(**********************Pointing************************)	
	(*ActAmbTemp_East:LREAL;
	ActAmbTemp_South:LREAL;
	AmbTempCorrVal_1:LREAL;
	AmbTempCorrVal_2:LREAL;
	TiltXRaw_One:LREAL;
	TiltYRaw_One:LREAL;
	TiltXArcsec_One:LREAL;
	TiltYArcsec_One: BOOL;
	TiltXFilt_One:LREAL;
	TiltYFilt_One:LREAL;
	TiltTemp_One:LREAL;
	TiltXRaw_Two:LREAL;
	TiltYRaw_Two:LREAL;
	TiltXArcsec_Two:LREAL;
	TiltYArcsec_Two: BOOL;
	TiltXFilt_Two:LREAL;
	TiltYFilt_Two:LREAL;
	TiltTemp_Two:LREAL;
	TiltCorrVal_Az:LREAL;
	TiltCorrVal_EL:LREAL;
	PmCorrVal_Az: BOOL;
	PmCorrVal_EL: BOOL;
	StaticCorrActive:BOOL;
	TiltCorrActive:BOOL;
	Pointing_TiltOn:UINT;
	TempCorrActive:BOOL;
	BandForCorr:UINT;*)
	Pointing_TiltOn:UINT;
(**************************Tracking********************************)
(*	tr_initOk:BOOL;(*Tracking function program is initialized and ready for operation*)
	tr_valid:BOOL;(*The tracking controller’s output is within the position ranges of the dish structure.*)
	tr_Table_error:BOOL;(*The table reports an error *)
	tr_obj_valid:BOOL;(*Tracking object has valid tracking data.*)
	tr_selFIy:BOOL;(*FIynomial tracking selected as source*)
	act_statOffset_value_Xel:LREAL;(*Actual azimuth static offset*)
	act_statOffset_value_El:LREAL;(*Elevation azimuth static offset*)
	p_desired_AZ:LREAL;(*Azimuth position output of the Tracking Controller*)
	p_desired_EL:LREAL;(*Elevation position output of the Tracking Controller*)
	tr_TimeRemaining:LREAL;(*Time till the last point in the track table is reached*)
	OnSourceDev:LREAL;(*Actual calculated “On Sky” rms tracking error.*) *)
(*********Read parameteers*******)
	AxRef:ARRAY[1..5] OF AXIS_REF;
	P_shape_value:ARRAY[1..5] OF LREAL;
	V_shape_value:ARRAY[1..5] OF LREAL;
	V_act_value:ARRAY[1..5] OF LREAL;
	r_write_position_az: LREAL; // Used internally for interpolator and pointing model calculations
    r_write_position_az_out: LREAL; (*the position written to the virvual azimuth axis*)
	r_write_position_el: LREAL; // Used internally for interpolator and pointing model calculations
    r_write_position_el_out: LREAL;(*the position written to the virvual elevation axis*)
	r_write_position_FI: LREAL;(*the position written to the virvual FeedIndexer axis*)
	r_write_position_FI_out: LREAL;(*the position written to the virvual FeedIndexer axis*)
	
END_VAR

VAR_GLOBAL RETAIN PERSISTENT
	R_total_distance_AZ:LREAL;
	R_total_distance_EL_deg:LREAL;
	R_total_distance_EL_m:LREAL;
	R_total_distance_FI:LREAL;
	
	LeapSecPTP: UINT :=37;    // Storage for Leap seconds 
	
END_VAR

// IndraMotionMlc1/Application/POUs/Motion/P_Position_and_MJD
(*The program is built for calculating the position of real axis, virtual axis and the MJD time,
and writing software limit of azimuth *)
PROGRAM P_Position_and_MJD
VAR
(*With the function block "MB_WriteRealParameter" you can write a defined value to the parameter belonging to the parameter number*)
	fb_write_negative_a: MB_WriteRealParameter;
	fb_write_negative_s: MB_WriteRealParameter;
	fb_write_positive_a: MB_WriteRealParameter;
	fb_write_positive_s: MB_WriteRealParameter;
(*the blink function block is for triggering MB_WriteRealParameter function block*)
	fb_blink_1: BLINK;
	fb_blink_2: BLINK;
	fb_blink_3: BLINK;
	fb_blink_4: BLINK;
(*the value is written to MB_WriteRealParameter*)
	r_negative_limit: REAL;
	r_positive_limit: REAL;
(*the elevation limit control*)
	fb_blink_diagnos_el: BLINK;
	fb_diagnose_el: MB_ReadStringParameter;
	str_diagnose_el: STRING;
	fb_blink_5: BLINK;
	fb_blink_6: BLINK;
	fb_write_negative_el: MB_WriteRealParameter;
	fb_write_positive_el: MB_WriteRealParameter;
	r_limit_el_up: REAL;
	r_limit_el_down: REAL;
	b_limit_up_el: BOOL;
	b_limit_down_el: BOOL;
	rtrig_set_limit_up: R_TRIG;
	rtrig_set_limit_down: R_TRIG;
	fb_blink_7: BLINK;
	fb_write_91_az1: MB_WriteRealParameter;
	fb_blink_8: BLINK;
	fb_blink_9: BLINK;
	fb_blink_10: BLINK;
	fb_blink_11: BLINK;
	fb_write_91_az2: MB_WriteRealParameter;
	fb_write_91_el1: MB_WriteRealParameter;
	fb_write_91_el2: MB_WriteRealParameter;
	fb_write_91_FI: MB_WriteRealParameter;
	fb_blink_12: BLINK;
	fb_write_91_FI2: MB_WriteRealParameter;
	r_pos_FI_1: REAL;
	i_counter_hr: BOOL;
	rtrig_hr:R_TRIG;
	
	fb_blink_111: BLINK;
	fb_write_negative_a_v: MB_WriteRealParameter;
	fb_blink_1_v: BLINK;
	fb_blink_2_v: BLINK;
	fb_write_negative_s_v: MB_WriteRealParameter;
	fb_blink_3_v: BLINK;
	fb_write_positive_a_v: MB_WriteRealParameter;
	
	temp_a:LREAL:=3135.4451;
	temp_b:LREAL:=3013.785;	
	temp_c:LREAL;
	r_pos_az_org :LREAL;
	r_pos_az_v_org :LREAL;
	r_pos_el_org:LREAL;
	r_pos_el_v_org:LREAL;

	fb_real_drive3_s51: MB_ReadRealParameter;
	r_pos_motor3_1: REAL;
	
	i_overlop:BOOL;
	rtrig_overlop:R_TRIG;
	
	
	DeltaB_temp: LREAL;
	
	B_TEMP: LREAL;
	
	MB_AxisDistanceAccumulator_2: MB_AxisDistanceAccumulator;
	bDisenable1: BOOL;
	test_1: LREAL;
	test_2: LREAL;
	test_old: LREAL;
	normal_count:DINT:=995;
	low_count:DINT:=9995;
	fast_count:DINT:=9995;
	i_change_sign_count:DINT;
	r_threshold:REAL;
END_VAR
VAR RETAIN
	r_last_position_az: REAL:=1;
	l_control:LREAL;
	a_control:REAL:=3035.4;
	b_control:REAL:=3035.1;
	b_motor_count:DINT:=0;
	b_sign_delay:BOOL:=0;
	b_sign_delay_count:DINT:=0;
	r_test_value:LREAL;
	i_test_value:DINT:=0;
	fb_read_source_code_3: MB_ReadParameter;
	r_source_code_3: DINT;
	r_source_to_elevation: LREAL;
END_VAR

 	//axisdata[7].rActualPosition_i;
r_source_to_elevation:=(DINT_TO_LREAL(r_source_code_3)/536870912)*360.0-64.812477;

	MB_AxisDistanceAccumulator_2(
	Enable:= bDisenable1, 
	TotalDistance:= 1000000, 
	InOperation=> , 
	Error=> , 
	ErrorID=> , 
	ErrorIdent=> , 
	DistanceReached=> , 
	AccumulatedDistance=> r_length_Distance_1, 
	Axis:= Drive3);
	
	IF	r_pos_motor3<0.01 AND r_pos_motor3>=0 THEN
	i_overlop:=TRUE;
	ELSE
	i_overlop:=FALSE;
	END_IF	
	rtrig_overlop(clk:=i_overlop);
	IF rtrig_overlop.Q=TRUE THEN
	b_motor_count:=b_motor_count+1;
	END_IF
		
	l_control:=SQRT(a_control*a_control+b_control*b_control-2*a_control*b_control*COS(deg2rad(112.0255-ML_Base.AxisData[3].rActualPosition_i)))-1151;
//	
//	temp_c:= SQRT(temp_a*temp_a + temp_b*temp_b-2*temp_a*temp_b*COS((115.5-r_pos_el_v)*3.1415926/180.0));
//	gear_ratio:=temp_a*temp_b*SIN((115.5-r_pos_el_v)*3.1415926/180.0)/temp_c*6.0*168.0/25.0/180.0*3.1415926;
	
	

(*<<time1<<<<<<<<<<<<<<<<<<<<<<<<<<<<<< real position of azimuth elevation and FeedIndexer>>>>>>>>>>>>>>>>>>>>>>>>>>>>>>>>*)
(*the azimuth position is judged by zone signal*)

	IF axisdata[1].Axis_Inbb=TRUE THEN	
		//r_pos_az_org:=axisdata[1].rActualPosition_i;
		//r_pos_az_1:=r_pos_az_org+C1+C3*SIN((r_pos_az_org-C4)*3.1415926/180)*TAN(r_pos_el_org*3.1415926/180)+C5*TAN(r_pos_el_org*3.1415926/180)+C6/COS(r_pos_el_org*3.1415926/180);		
	//	r_pos_az_modify:=r_pos_az_1;
	    r_pos_az_modify:=axisdata[1].rActualPosition_i;
		IF r_pos_az_1>=360.0 THEN 
			r_pos_az_modify:=r_pos_az_1-360.00;
		END_IF
		IF r_pos_az_1<0.0 THEN 
			r_pos_az_modify:=r_pos_az_1+360.00;
		END_IF
			
	END_IF;		
		(*IF b_zone_az=FALSE AND axisdata[1].rActualPosition_i>75 AND axisdata[1].rActualPosition_i<360 THEN
			r_pos_az:=axisdata[1].rActualPosition_i-360;
			r_pos_az_v:=axisdata[1].rActualPosition_i-360;
//		ELSIF axisdata[1].rActualPosition_i>299 THEN
	//		r_pos_az:=axisdata[1].rActualPosition_i-360;
//			r_pos_az_v:=axisdata[1].rActualPosition_i-360;
        ELSE
        r_pos_az:=axisdata[1].rActualPosition_i;
		r_pos_az_v:=axisdata[1].rActualPosition_i;
		END_IF;*)
        r_pos_az:=axisdata[1].rActualPosition_i;
		r_pos_az_v:=axisdata[7].rActualPosition_i;
	//	END_IF;
   IF gc_b_sim_on THEN
	IF ABS (r_pos_az_v ) = 360 THEN	
	r_pos_az:=0.0000;
	r_pos_az_v := 0.0000;
	END_IF
   END_IF
	
	//angleerror := axisdata[1].rActualPosition_i - axisdata[2].rActualPosition_i;

	AZ_encoder_last:=r_pos_az_v;
	
	IF axisdata[5].rActualPosition_i < 180 THEN
		r_pos_Fi:=axisdata[5].rActualPosition_i;
	    r_pos_Fi_v:=axisdata[5].rActualPosition_i;
	ELSE
		r_pos_Fi:=axisdata[5].rActualPosition_i-360;
	    r_pos_Fi_v:=axisdata[5].rActualPosition_i-360;
	END_IF
	FI_encoder_last:=r_pos_fi_v;
	
//r_pos_el_org:=axisdata[3].rActualPosition_i;
//r_pos_el_1:=r_pos_el_org+C2+C3*COS((r_pos_az_org-C4)*3.1415926/180)+C7*COS(r_pos_el_org*3.1415926/180)+0;	
//r_pos_el_modify	:=r_pos_el_1;
r_pos_el:=axisdata[3].rActualPosition_i;
//r_pos_el:=r_source_to_elevation;
r_pos_el_v:=axisdata[3].rActualPosition_i;
(* From SKA063 project
r_pos_el:=ML_Base.AxisData[11].rActualPosition_i;
r_pos_el_v:=ML_Base.AxisData[11].rActualPosition_i; *)

(*<<<<<<<<<<<<<<<<<<<<<<<<<<<<<<<<<<<<<<<<<<<<<<<<<<<calculation for MJD >>>>>>>>>>>>>>>>>>>>>>>>>>>>>>>>>>>>>>>*)
(*the definition of MJD is shown in the global variables*)
(*the module of v_time_master axis is 360,so that it take 6minuts to run one cycle*)
IF	axisdata[10].rActualPosition_i<0.01 AND axisdata[10].rActualPosition_i>=0 THEN
	i_counter_hr:=TRUE;
ELSE
	i_counter_hr:=FALSE;
END_IF	
rtrig_hr(clk:=i_counter_hr);
IF rtrig_hr.Q=TRUE THEN
	i_num_quarter:=i_num_quarter+1;
END_IF
IF i_num_quarter=240 THEN
	i_num_quarter:=0;
	di_MJD_day:=di_MJD_day+1;
END_IF

//lr_MJD_current:=TO_REAL(di_MJD_day)+(360*TO_REAL(i_num_quarter)+axisdata[10].rActualPosition_i)/86400+1.0/3.0; // Sets MJD to Beijing time
lr_MJD_current:=TO_REAL(di_MJD_day)+(360*TO_REAL(i_num_quarter)+axisdata[10].rActualPosition_i)/86400;
lr_TAIoffset_current:= (lr_MJD_Current-gc_SKAEpochMJD)*86400+(time_cds.Status.LeapSecPTP); // Minus 10s if you want to correlate to a unix timestamp


(*<<<<<<<<<<<<<<<<<calculate the following error of trajectory>>>>>>>>>>>>>>>>>>>*)

IF ABS(r_vel_EL)>=0.5 THEN
	r_threshold:=0.25;
ELSE 
	r_threshold:=0.15;
END_IF

IF b_open_channel_az AND b_open_channel_el THEN
//IF ABS(lr_MJD_current-track_table[i_start].MJD-0.0000000254)*86400<=0.0005 AND b_sign_delay=0 THEN
	IF ABS(lr_TAIoffset_current-track_table[i_start].TAIoffset-0.0022)<=0.0005 AND b_sign_delay=0 THEN
	b_sign_delay:=1;
//	r_test_value:=0;
	i_test_value:=0;
	r_track_error[1]:=track_table[i_start].Azimuth-r_pos_az;
	
(*   For Elevation orientation axis

	r_track_error[2]:=track_table[i_start].Elevation_ori+r_offset_el_program-r_pos_el;
   IF ABS(r_track_error[2])<r_threshold THEN
		test_1:=Encoder_to_motor(track_table[i_start].Elevation_ori)-Encoder_to_motor(track_table[i_start].Elevation_ori-r_track_error[2]);
		test_2:=Encoder_to_motor(track_table[i_start].Elevation_ori)-Encoder_to_motor(track_table[i_start].Elevation_ori+r_track_error[2]);
//		test_3:=test_1+test_old;
	ELSE
		test_1:=0;
		test_2:=0;
		r_compensation_abs:=0;
		test_old:=0;
	END_IF *)
	
END_IF
	IF b_sign_delay =1 THEN

	i_test_value:=i_test_value+1;
	
	IF i_test_value>995 THEN 
		r_test_value:=r_compensation_abs;
	ELSE
		r_test_value:=r_compensation_abs+test_1/995;
	END_IF
		r_compensation_abs:=r_test_value;
		
	END_IF
		
	END_IF

IF b_sign_delay =1 THEN 
	b_sign_delay_count:=b_sign_delay_count+1;
END_IF

IF ABS(r_vel_EL)<0.002 THEN
	i_change_sign_count:=9995;
ELSIF ABS(r_vel_EL)>0.6 AND ABS(r_vel_EL)<0.8 THEN
	i_change_sign_count:=9995;
ELSIF ABS(r_vel_EL)>=0.8 THEN
	i_change_sign_count:=12995;	
ELSE 
	i_change_sign_count:=normal_count;	
END_IF




IF b_sign_delay_count>i_change_sign_count THEN
	b_sign_delay_count:=0;
	b_sign_delay:=0;
END_IF




IF b_off_write=TRUE THEN
	r_limit_s91:=11;
ELSE
	r_limit_s91:=1.4;
END_IF;
(*<<<<<<<<<<<<<<<<<<the azimuth limit control>>>>>>>>>>>>>>>>>>>>*)
IF (r_pos_az<-250) OR (r_pos_az>250) THEN
(*the range of azimuth is -179~359*)
	//r_negative_limit:=89;
	//r_positive_limit:=271;
	r_negative_limit:=-275;
	r_positive_limit:=275;
ELSE
	//r_negative_limit:=0;
	//r_positive_limit:=360;
	r_negative_limit:=-275;
	r_positive_limit:=275;
END_IF;
(*
(*<<<<<<<<<<<<<<<<<<<<<<<<<the elevation limit control>>>>>>>>>>>>>>>>>>>>>>>*)
IF str_diagnose_el='F6029 ' THEN
	b_limit_up_el:=TRUE;
ELSE
	b_limit_up_el:=FALSE;
END_IF
rtrig_set_limit_up(clk:=b_limit_up_el);
IF rtrig_set_limit_up.Q=TRUE THEN
	r_limit_el_up:=90.05;
END_IF
IF r_pos_el <=90.1 THEN
	r_limit_el_up:=90.15;
END_IF

IF str_diagnose_el='F6030 ' THEN
	b_limit_down_el:=TRUE;
ELSE
	b_limit_down_el:=FALSE;
END_IF
rtrig_set_limit_down(clk:=b_limit_down_el);
IF rtrig_set_limit_down.Q=TRUE THEN
	r_limit_el_down:=14.7;
END_IF
IF r_pos_el >=14.65 THEN
	r_limit_el_down:=14.6;
END_IF
*)



//P_Position_and_MJD.A_Write_Limit_Value();lr_TAIoffset_current
//Time Sensitive pointing data
Time_cds.Status.TAIOffset:=lr_TAIoffset_current;
IF gc_b_sim_on THEN 
	IF r_pos_az = -360 THEN
		r_pos_az:= 0;
	END_IF

END_IF

Azimuth.Status.p_Act:=pointing.Status.TotalPointCorr_Az/gc_lr_arcsec2deg+r_pos_az;
Azimuth.Status.p_Enc:=r_pos_az;
Elevation.Status.p_Act:=pointing.Status.TotalPointCorr_El/gc_lr_arcsec2deg+r_pos_el;
Elevation.Status.p_Enc:=r_pos_el;

Pointing.Status.CurrentPointing[0]:= Time_cds.Status.TAIoffset;
Pointing.Status.CurrentPointing[1]:= Azimuth.Status.p_Act;
Pointing.Status.CurrentPointing[2]:= Elevation.Status.p_Act;
Pointing.Status.CurrentPointing[3]:= Azimuth.Status.p_Enc;
Pointing.Status.CurrentPointing[4]:= Elevation.Status.p_Enc;
Pointing.Status.CurrentPointing[5]:= pointing.Status.TiltCorrVal_Az;
Pointing.Status.CurrentPointing[6]:= pointing.Status.TiltCorrVal_El;

ACTION A_Write_Limit_Value:
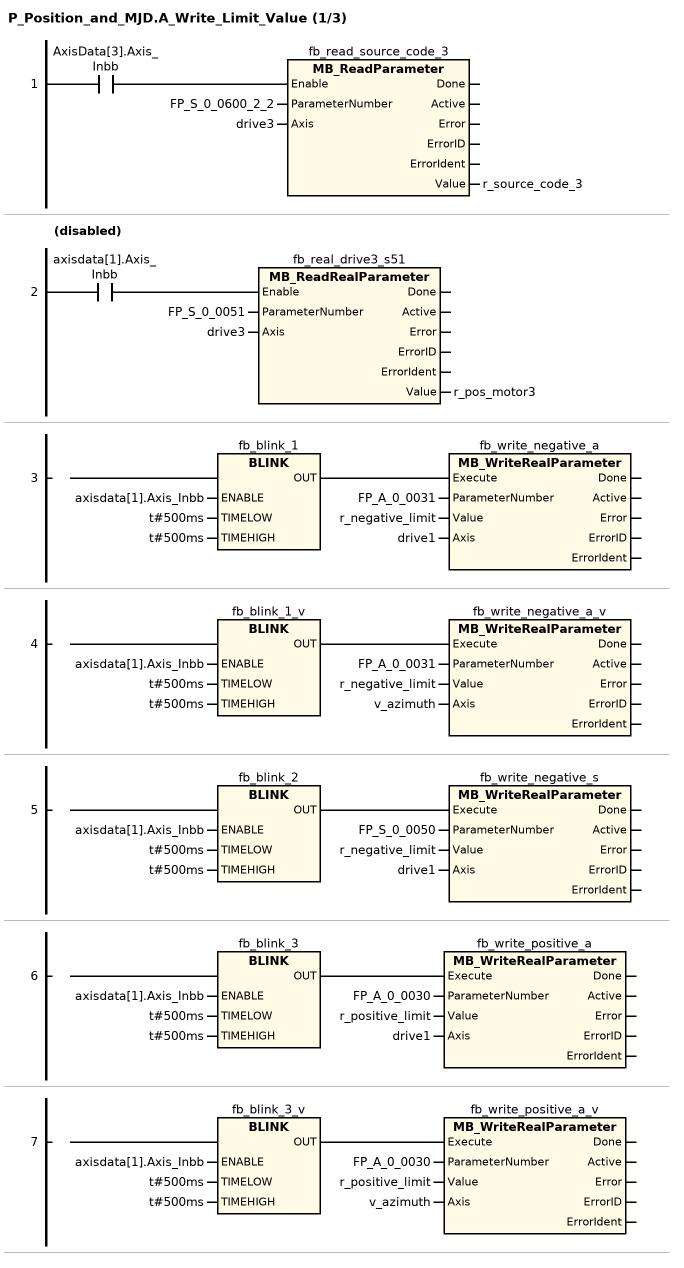
// NETWORK 1
fb_read_source_code_3(
    Enable := AxisData[3].Axis_Inbb,
    ParameterNumber := FP_S_0_0600_2_2,
    Axis := drive3,
    Value => r_source_code_3); // MB_ReadParameter

// NETWORK 2 (disabled)
//   FP_S_0_0051: Position limit value, negative
//   drive3: the value is written to MB_WriteRealParameter
// fb_real_drive3_s51(
//     Enable := axisdata[1].Axis_Inbb,
//     ParameterNumber := FP_S_0_0051,
//     Axis := drive3,
//     Value => r_pos_motor3); // MB_ReadRealParameter

// NETWORK 3
//   fb_write_negative_a: With the function block "MB_WriteRealParameter" you can write a defined value to the parameter belonging to the parameter number
//   fb_blink_1: the blink function block is for triggering MB_WriteRealParameter function block
//   axisdata[1].Axis_Inbb: A-0-0021.13 -RD- Axis is ready for power to the amplifier (bb)
//   FP_A_0_0031: Position limit value, negative
//   r_negative_limit: the value is written to MB_WriteRealParameter
//   drive1: Real axis "Drive1" with axis number 1
fb_blink_1(ENABLE := axisdata[1].Axis_Inbb, TIMELOW := t#500ms, TIMEHIGH := t#500ms); // BLINK
fb_write_negative_a(
    Execute := fb_blink_1.OUT,
    ParameterNumber := FP_A_0_0031,
    Value := r_negative_limit,
    Axis := drive1); // MB_WriteRealParameter

// NETWORK 4
//   axisdata[1].Axis_Inbb: A-0-0021.13 -RD- Axis is ready for power to the amplifier (bb)
//   FP_A_0_0031: Position limit value, negative
//   r_negative_limit: the value is written to MB_WriteRealParameter
//   v_azimuth: Virtual axis "v_azimuth" with axis number 7
fb_blink_1_v(ENABLE := axisdata[1].Axis_Inbb, TIMELOW := t#500ms, TIMEHIGH := t#500ms); // BLINK
fb_write_negative_a_v(
    Execute := fb_blink_1_v.OUT,
    ParameterNumber := FP_A_0_0031,
    Value := r_negative_limit,
    Axis := v_azimuth); // MB_WriteRealParameter

// NETWORK 5
//   axisdata[1].Axis_Inbb: A-0-0021.13 -RD- Axis is ready for power to the amplifier (bb)
//   FP_S_0_0050: Negative position limit value
//   r_negative_limit: the value is written to MB_WriteRealParameter
//   drive1: Real axis "Drive1" with axis number 1
fb_blink_2(ENABLE := axisdata[1].Axis_Inbb, TIMELOW := t#500ms, TIMEHIGH := t#500ms); // BLINK
fb_write_negative_s(
    Execute := fb_blink_2.OUT,
    ParameterNumber := FP_S_0_0050,
    Value := r_negative_limit,
    Axis := drive1); // MB_WriteRealParameter

// NETWORK 6
//   axisdata[1].Axis_Inbb: A-0-0021.13 -RD- Axis is ready for power to the amplifier (bb)
//   FP_A_0_0030: Position limit value, positive
//   drive1: Real axis "Drive1" with axis number 1
fb_blink_3(ENABLE := axisdata[1].Axis_Inbb, TIMELOW := t#500ms, TIMEHIGH := t#500ms); // BLINK
fb_write_positive_a(
    Execute := fb_blink_3.OUT,
    ParameterNumber := FP_A_0_0030,
    Value := r_positive_limit,
    Axis := drive1); // MB_WriteRealParameter

// NETWORK 7
//   axisdata[1].Axis_Inbb: A-0-0021.13 -RD- Axis is ready for power to the amplifier (bb)
//   FP_A_0_0030: Position limit value, positive
//   v_azimuth: Virtual axis "v_azimuth" with axis number 7
fb_blink_3_v(ENABLE := axisdata[1].Axis_Inbb, TIMELOW := t#500ms, TIMEHIGH := t#500ms); // BLINK
fb_write_positive_a_v(
    Execute := fb_blink_3_v.OUT,
    ParameterNumber := FP_A_0_0030,
    Value := r_positive_limit,
    Axis := v_azimuth); // MB_WriteRealParameter

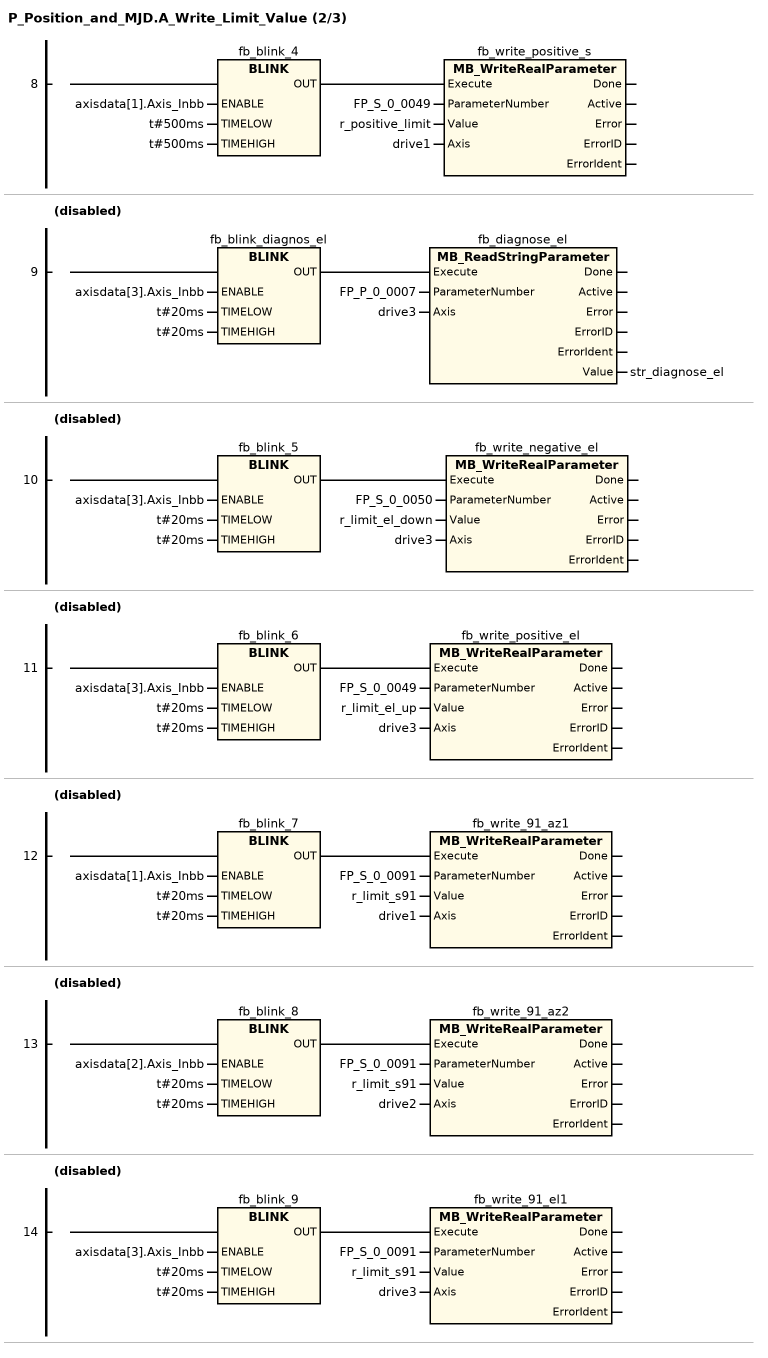
// NETWORK 8
//   axisdata[1].Axis_Inbb: A-0-0021.13 -RD- Axis is ready for power to the amplifier (bb)
//   FP_S_0_0049: Positive position limit value
//   drive1: Real axis "Drive1" with axis number 1
fb_blink_4(ENABLE := axisdata[1].Axis_Inbb, TIMELOW := t#500ms, TIMEHIGH := t#500ms); // BLINK
fb_write_positive_s(
    Execute := fb_blink_4.OUT,
    ParameterNumber := FP_S_0_0049,
    Value := r_positive_limit,
    Axis := drive1); // MB_WriteRealParameter

// NETWORK 9 (disabled)
//   fb_blink_diagnos_el: the elevation limit control
//   axisdata[3].Axis_Inbb: A-0-0021.13 -RD- Axis is ready for power to the amplifier (bb)
//   FP_P_0_0007: Display text of diagnostic message
//   drive3: Real axis "Drive3" with axis number 3
// fb_blink_diagnos_el(ENABLE := axisdata[3].Axis_Inbb, TIMELOW := t#20ms, TIMEHIGH := t#20ms); // BLINK
// fb_diagnose_el(
//     Execute := fb_blink_diagnos_el.OUT,
//     ParameterNumber := FP_P_0_0007,
//     Axis := drive3,
//     Value => str_diagnose_el); // MB_ReadStringParameter

// NETWORK 10 (disabled)
//   axisdata[3].Axis_Inbb: A-0-0021.13 -RD- Axis is ready for power to the amplifier (bb)
//   FP_S_0_0050: Negative position limit value
//   drive3: Real axis "Drive3" with axis number 3
// fb_blink_5(ENABLE := axisdata[3].Axis_Inbb, TIMELOW := t#20ms, TIMEHIGH := t#20ms); // BLINK
// fb_write_negative_el(
//     Execute := fb_blink_5.OUT,
//     ParameterNumber := FP_S_0_0050,
//     Value := r_limit_el_down,
//     Axis := drive3); // MB_WriteRealParameter

// NETWORK 11 (disabled)
//   axisdata[3].Axis_Inbb: A-0-0021.13 -RD- Axis is ready for power to the amplifier (bb)
//   FP_S_0_0049: Positive position limit value
//   drive3: Real axis "Drive3" with axis number 3
// fb_blink_6(ENABLE := axisdata[3].Axis_Inbb, TIMELOW := t#20ms, TIMEHIGH := t#20ms); // BLINK
// fb_write_positive_el(
//     Execute := fb_blink_6.OUT,
//     ParameterNumber := FP_S_0_0049,
//     Value := r_limit_el_up,
//     Axis := drive3); // MB_WriteRealParameter

// NETWORK 12 (disabled)
//   axisdata[1].Axis_Inbb: A-0-0021.13 -RD- Axis is ready for power to the amplifier (bb)
//   FP_S_0_0091: Bipolar velocity limit value
//   drive1: Real axis "Drive1" with axis number 1
// fb_blink_7(ENABLE := axisdata[1].Axis_Inbb, TIMELOW := t#20ms, TIMEHIGH := t#20ms); // BLINK
// fb_write_91_az1(
//     Execute := fb_blink_7.OUT,
//     ParameterNumber := FP_S_0_0091,
//     Value := r_limit_s91,
//     Axis := drive1); // MB_WriteRealParameter

// NETWORK 13 (disabled)
//   axisdata[2].Axis_Inbb: A-0-0021.13 -RD- Axis is ready for power to the amplifier (bb)
//   FP_S_0_0091: Bipolar velocity limit value
//   drive2: Real axis "Drive2" with axis number 2
// fb_blink_8(ENABLE := axisdata[2].Axis_Inbb, TIMELOW := t#20ms, TIMEHIGH := t#20ms); // BLINK
// fb_write_91_az2(
//     Execute := fb_blink_8.OUT,
//     ParameterNumber := FP_S_0_0091,
//     Value := r_limit_s91,
//     Axis := drive2); // MB_WriteRealParameter

// NETWORK 14 (disabled)
//   axisdata[3].Axis_Inbb: A-0-0021.13 -RD- Axis is ready for power to the amplifier (bb)
//   FP_S_0_0091: Bipolar velocity limit value
//   drive3: Real axis "Drive3" with axis number 3
// fb_blink_9(ENABLE := axisdata[3].Axis_Inbb, TIMELOW := t#20ms, TIMEHIGH := t#20ms); // BLINK
// fb_write_91_el1(
//     Execute := fb_blink_9.OUT,
//     ParameterNumber := FP_S_0_0091,
//     Value := r_limit_s91,
//     Axis := drive3); // MB_WriteRealParameter

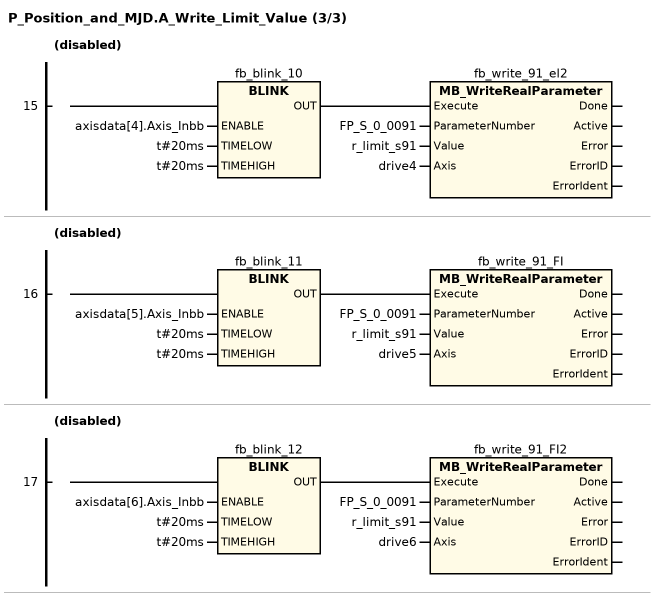
// NETWORK 15 (disabled)
//   axisdata[4].Axis_Inbb: A-0-0021.13 -RD- Axis is ready for power to the amplifier (bb)
//   FP_S_0_0091: Bipolar velocity limit value
//   drive4: Real axis "Drive4" with axis number 4
// fb_blink_10(ENABLE := axisdata[4].Axis_Inbb, TIMELOW := t#20ms, TIMEHIGH := t#20ms); // BLINK
// fb_write_91_el2(
//     Execute := fb_blink_10.OUT,
//     ParameterNumber := FP_S_0_0091,
//     Value := r_limit_s91,
//     Axis := drive4); // MB_WriteRealParameter

// NETWORK 16 (disabled)
//   axisdata[5].Axis_Inbb: A-0-0021.13 -RD- Axis is ready for power to the amplifier (bb)
//   FP_S_0_0091: Bipolar velocity limit value
//   drive5: Real axis "Drive5" with axis number 5
// fb_blink_11(ENABLE := axisdata[5].Axis_Inbb, TIMELOW := t#20ms, TIMEHIGH := t#20ms); // BLINK
// fb_write_91_FI(
//     Execute := fb_blink_11.OUT,
//     ParameterNumber := FP_S_0_0091,
//     Value := r_limit_s91,
//     Axis := drive5); // MB_WriteRealParameter

// NETWORK 17 (disabled)
//   axisdata[6].Axis_Inbb: A-0-0021.13 -RD- Axis is ready for power to the amplifier (bb)
//   FP_S_0_0091: Bipolar velocity limit value
//   drive6: Real axis "Drive6" with axis number 6
// fb_blink_12(ENABLE := axisdata[6].Axis_Inbb, TIMELOW := t#20ms, TIMEHIGH := t#20ms); // BLINK
// fb_write_91_FI2(
//     Execute := fb_blink_12.OUT,
//     ParameterNumber := FP_S_0_0091,
//     Value := r_limit_s91,
//     Axis := drive6); // MB_WriteRealParameter
END_ACTION

END_PROGRAM

// IndraMotionMlc1/Application/POUs/TCP/Message/deg2rad
FUNCTION deg2rad : LREAL
VAR_INPUT
degree_in:LREAL;	
END_VAR
VAR
END_VAR

deg2rad:=degree_in/180.0*3.1415926;

END_FUNCTION

// IndraMotionMlc1/Application/POUs/TCP/Message/Encoder_to_motor
FUNCTION Encoder_to_motor : LREAL
VAR_INPUT
	encoder_input:LREAL;
END_VAR
VAR
END_VAR

(*
Encoder_to_motor:=P1*EXPT(encoder_input+40,8)+P2*EXPT(encoder_input+40,7)+P3*EXPT(encoder_input+40,6)+P4*EXPT(encoder_input+40,5)
					+P5*EXPT(encoder_input+40,4)+P6*EXPT(encoder_input+40,3)+P7*EXPT(encoder_input+40,2)
						+P8*(encoder_input+40)+P9+1000000;
*)						
(*Encoder_to_motor:=P1*EXPT(encoder_input,9)+P2*EXPT(encoder_input,8)+P3*EXPT(encoder_input,7)+P4*EXPT(encoder_input,6)
					+P5*EXPT(encoder_input,5)+P6*EXPT(encoder_input,4)+P7*EXPT(encoder_input,3)+P8*EXPT(encoder_input,2)
						+P9*(encoder_input)+P10;
*)
					
Encoder_to_motor:=P1*EXPT(encoder_input,9)+P2*EXPT(encoder_input,8)+P3*EXPT(encoder_input,7)+P4*EXPT(encoder_input,6)
					+P5*EXPT(encoder_input,5)+P6*EXPT(encoder_input,4)+P7*EXPT(encoder_input,3)+P8*EXPT(encoder_input,2)
						+P9*(encoder_input)+P10-5441.92821;

END_FUNCTION

// IndraMotionMlc1/Application/POUs/Motion/P_EL_VEL_MODE
PROGRAM P_EL_VEL_MODE
VAR
		(*******variable of the velocity control*******)
	
	Vmax_EL:LREAL:=1.4;
	Aacc_EL:LREAL:=0.6;
	Adec_EL:LREAL:=0.6;
	
	Pos_EL_current:LREAL;
	
	V_acc_EL:LREAL;
	V_dec_EL:LREAL;
	
	V_last_EL:LREAL;
	T_period_EL:LREAL:=0.001;
	Pos_EL_closeloop_error:LREAL:=1.0;
(**********第一种丝杠参数（旧丝杠）************)	
(*	A1:REAL:= 1.301E-13;
	A2:REAL:=-4.148E-11 ;
	A3:REAL:=4.854E-09;
	A4:REAL:=-2.212E-07 ;
	A5:REAL:=-1.601E-06;
	A6:REAL:= 0.0005281 ;
	A7:REAL:= -0.02546 ;
	A8:REAL:=1.926;
	A9:REAL:= 115.6;
*)	
(**********第二种丝杠参数（新丝杠）************)	
	A1:REAL:= -4.201E-13;
	A2:REAL:=1.683E-10 ;
	A3:REAL:=-2.855E-08;
	A4:REAL:=2.674E-06 ;
	A5:REAL:=-0.0001496;
	A6:REAL:= 0.004967 ;
	A7:REAL:= -0.09779 ;
	A8:REAL:=2.78;
	A9:REAL:= 145.2;	

	
	
	v_pos_calculate:LREAL;		
	(*******End variable of the velocity control*******)
	V_command_EL1: LREAL;
	
	T_sum_goto:LREAL;
	T_sum_goto_ratio:LREAL;
	
END_VAR

(**************EL Velocity control mode ***************)
(********************第二个丝杠的减速比*********************)
IF r_pos_el > 14 THEN
	K_gear_ratio:=(A1*EXPT(r_pos_el,8)+A2*EXPT(r_pos_el,7)+A3*EXPT(r_pos_el,6)+A4*EXPT(r_pos_el,5)
					+A5*EXPT(r_pos_el,4)+A6*EXPT(r_pos_el,3)+A7*EXPT(r_pos_el,2)+A8*r_pos_el
						+A9)*10;
						
END_IF
						
						
V_max_vel_motor:=Vmax_EL*K_gear_ratio;						
(**************EL Velocity control mode ***************)
IF b_scc_goto OR b_track_on THEN 
Pos_EL_current:=r_pos_el;
	IF b_scc_goto THEN
		IF r_pos_el<30 AND ABS(r_goto_el_I-r_pos_el)>0.02 THEN		
			m_dKa:=0.75;
			m_dKv:=0.08;
		ELSE
			m_dKa:=0.75;
			m_dKv:=0.08;
		END_IF

	(*IF ABS(r_goto_el_I-r_EL_current_when_goto_cmd)<1.1 THEN
		T_sum_goto:=4.5;
	ELSIF 9.5<ABS(r_goto_el_I-r_EL_current_when_goto_cmd) AND ABS(r_goto_el_I-r_EL_current_when_goto_cmd)<10.1 THEN
		T_sum_goto:=11.5;	
	ELSE
		//T_sum_goto:=ABS(r_goto_el_I-r_EL_current_when_goto_cmd)/1.4+1;
		T_sum_goto:=ABS(r_goto_el_I-r_EL_current_when_goto_cmd)/1.4+1;
			IF T_sum_goto<4.5 THEN
				T_sum_goto:=4.5;
			END_IF
	END_IF*)
	
	IF ABS(r_goto_el_I-r_EL_current_when_goto_cmd)<1.1 THEN
		T_sum_goto:=4.5;
	ELSIF ABS(r_goto_el_I-r_EL_current_when_goto_cmd)<9.5 THEN
		T_sum_goto:=ABS(r_goto_el_I-r_EL_current_when_goto_cmd)*0.78+3.642;
	ELSIF ABS(r_goto_el_I-r_EL_current_when_goto_cmd)<10.1 THEN
		T_sum_goto:=11.5;
	ELSE
		//T_sum_goto:=ABS(r_goto_el_I-r_EL_current_when_goto_cmd)/1.4+1;
		T_sum_goto:=ABS(r_goto_el_I-r_EL_current_when_goto_cmd)*1.15-0.115;
			IF T_sum_goto<4.5 THEN
				T_sum_goto:=4.5;
			END_IF
	END_IF
	
	T_count_goto:=(T_count_goto+0.001);
	T_sum_goto_ratio:=T_count_goto/T_sum_goto;
	IF T_count_goto>=T_sum_goto THEN
		T_count_goto:=T_sum_goto;
		b_step_running_el:=0;
	END_IF
	Pos_EL_Aim:=F_cyclic_position(r_EL_current_when_goto_cmd,r_goto_el_I,0,0,0,0,T_sum_goto,T_sum_goto_ratio);	
//	Pos_EL_Aim:=r_goto_el_I;
	Pos_EL_error:=Pos_EL_Aim-Pos_EL_current;
		IF b_SCC_goto THEN
			r_following_3:=Pos_EL_error;
		END_IF	
	END_IF
	
	IF b_track_on THEN
	Pos_EL_Aim:=r_write_position_el;	
	Pos_EL_error:=Pos_EL_Aim-Pos_EL_current;

		IF r_pos_el <30 THEN 	
			IF ABS(Pos_EL_error)>0.02 THEN
			m_dKa:=0.75;
			m_dKv:=0.08;
			ELSE
			m_dKa:=0.75;
			m_dKv:=0.08;
			END_IF
		ELSE
			IF ABS(Pos_EL_error)>0.02 THEN
				m_dKa:=0.75;
				m_dKv:=0.08;
			ELSE
				m_dKa:=0.75;
				m_dKv:=0.08;
			END_IF
		END_IF
	END_IF


IF Pos_EL_error>=0 THEN
	V_acc_EL:=V_LastSpeed+Aacc_EL*T_period_EL*K_gear_ratio;
ELSE
	V_acc_EL:=V_LastSpeed-Aacc_EL*T_period_EL*K_gear_ratio;
END_IF
IF V_acc_EL>=Vmax_EL*K_gear_ratio THEN
	 V_acc_EL:=Vmax_EL*K_gear_ratio;
END_IF
IF V_acc_EL<=-Vmax_EL*K_gear_ratio THEN
	 V_acc_EL:=-Vmax_EL*K_gear_ratio;
END_IF

V_dec_EL:=SQRT(2*ABS(Pos_EL_error)*Adec_EL)*K_gear_ratio;
IF Pos_EL_error<0 THEN
	V_dec_EL:=-V_dec_EL;
END_IF

IF ABS(V_acc_EL)>=ABS(V_dec_EL) THEN
	V_command_EL:=V_dec_EL;
ELSE
	V_command_EL:=V_acc_EL;
END_IF

IF ABS(Pos_EL_error)<=Pos_EL_closeloop_error THEN
//	v_pos_calculate:=P_close_loop(Pos_EL_error);	
	V_command_EL:=P_close_loop(Pos_EL_error)+1.0*r_cyclic_velocity*K_gear_ratio;
//	V_command_EL:=P_close_loop(Pos_EL_error);
	V_command_EL1:=P_close_loop(Pos_EL_error)/K_gear_ratio;
//		m_dAUnsub2 := m_dAUnsub1;
//		m_dAUnsub1 := V_command_EL;
//		m_dAEnsub2 := m_dAEnsub1;
//		m_dAEnsub1 := Pos_EL_error;
//	V_command_EL:=P_close_loop(Pos_EL_error)*0.1*K_gear_ratio;
ELSE	
	V_LastOutput:=V_command_EL;	
END_IF
	V_LastSpeed:=V_command_EL;
END_IF

END_PROGRAM

// IndraMotionMlc1/Application/POUs/TCP/Message/F_cyclic_position
FUNCTION F_cyclic_position : LREAL
VAR_INPUT
	Pos_start:LREAL;
	pos_end:LREAL;
	vel_start:LREAL;
	vel_end:LREAL;
	acc_start:LREAL;
	acc_end:LREAL;
	T_sum:LREAL;
	T_count:LREAL;
END_VAR
VAR
	C0:LREAL;
	C1:LREAL;
	C2:LREAL;
	C3:LREAL;
	C4:LREAL;
	C5:LREAL;
	Y0:LREAL;
	Y1:LREAL;
	Y2:LREAL;
	Y3:LREAL;
	Y4:LREAL;
	Y5:LREAL;
	test:LREAL;
	
END_VAR

Y0:=Pos_start;
Y1:=vel_start*T_sum;
Y2:=acc_start*T_sum*T_sum/2;
Y3:=pos_end;
Y4:=vel_end*T_sum;
Y5:=acc_end*T_sum*T_sum/2;

C0:=Y0;
C1:=Y1;
C2:=Y2;
C3:=10*Y3-4*Y4+Y5-10*C0-6*C1-3*C2;
C4:=5*Y3-Y4-5*C0-4*C1-3*C2-2*C3;
C5:=Y3-C0-C1-C2-C3-C4;


F_cyclic_position:=C5*EXPT(T_count,5)+C4*EXPT(T_count,4)+C3*EXPT(T_count,3)+C2*EXPT(T_count,2)+C1*T_count+C0;
r_cyclic_velocity:=(5*C5*EXPT(T_count,4)+4*C4*EXPT(T_count,3)+3*C3*EXPT(T_count,2)+2*C2*EXPT(T_count,1)+C1)/T_sum;
test:=F_cyclic_position;

END_FUNCTION

// IndraMotionMlc1/Application/POUs/TCP/Message/P_CLOSE_LOOP
FUNCTION P_CLOSE_LOOP : LREAL
VAR_INPUT
	dError:LREAL;
END_VAR
VAR
	dspeed:LREAL:=0;
	MAIN_TIMER:LREAL:=0.001;
	(****calculate the K parameters*****)
(****1.0.    1.0****)	
//	m_dKp:REAL:=1.41443;
//	m_dTi:REAL:=1.41443;	
(****0.5.    1.0****)	
//	m_dKp:REAL:=1.00015;
//	m_dTi:REAL:=2.0003;	
(****0.3.    1.0****)	
//	m_dKp:REAL:=0.774714;
//	m_dTi:REAL:=2.58238;	
(****0.2.    1.0****)	
//	m_dKp:REAL:=0.632551;
//	m_dTi:REAL:=3.16276;
(****0.5.    0.1****)	
//	m_dKp:REAL:=10.0015;
//	m_dTi:REAL:=2.0003;
	(****0.3.    0.1****)	
	m_dKp:LREAL:=7.74714;
	m_dTi:LREAL:=2.58238;
		(****1.0.    0.1****)	
//	m_dKp:REAL:=14.1443;
//	m_dTi:REAL:=1.41443;
	(****0.2.    0.1****)	
//	m_dKp:REAL:=6.32551;
//	m_dTi:REAL:=3.16276;
	
	
	m_dKzn:LREAL:=0.707;	
	m_dA1:LREAL:=1.9874;
	m_dA2:LREAL:=-0.9874;
	m_dB0:LREAL:=0;
	m_dB1:LREAL:=0.08232;
	m_dB2:LREAL:=-0.08232;
	
END_VAR

	m_dTi:=1/0.707/SQRT(m_dKa);
	m_dKp:=m_dKa/m_dKv*m_dTi;

	IF V_LastOutput >= V_max_vel_motor THEN
		IF dError > 0 THEN
			dIntegralSpeed := m_dLastIntegral;
		ELSE
			dIntegralSpeed :=m_dLastIntegral + m_dKp * ( MAIN_TIMER / m_dTi) * dError;
		end_if
	ELSIF V_LastOutput<=-V_max_vel_motor THEN
		IF dError < 0 THEN
			dIntegralSpeed := m_dLastIntegral;
		ELSE
			dIntegralSpeed := m_dLastIntegral + m_dKp * (MAIN_TIMER / m_dTi) * dError;
		end_if
	ELSE
		r_Integral_thistime:=m_dKp * (MAIN_TIMER / m_dTi) * dError;
		dIntegralSpeed := m_dLastIntegral + m_dKp * (MAIN_TIMER / m_dTi) * dError;
	END_IF
	
	m_dLastIntegral := dIntegralSpeed;
	dspeed:=(dError * m_dKp + dIntegralSpeed)*0.1*K_gear_ratio;
	
	IF dspeed >= V_max_vel_motor THEN
		dspeed := V_max_vel_motor;
	ELSIF dspeed <= -V_max_vel_motor THEN
		dspeed := -V_max_vel_motor;
	END_IF
	V_LastOutput:=dspeed;
	P_CLOSE_LOOP:=dspeed;
(*	
	dspeed := m_dA1 * m_dAUnsub1 + m_dA2 * m_dAUnsub2+m_dB0 * dError + m_dB1 * m_dAEnsub1 + m_dB2 * m_dAEnsub2;
	m_dAUnsub2:=m_dAUnsub1;
	m_dAUnsub1:=dSpeed;
	
	m_dAEnsub2:=m_dAEnsub1;
	m_dAEnsub1:=dError;
	P_CLOSE_LOOP:=dspeed;
	*)

END_FUNCTION

// IndraMotionMlc1/Application/POUs/Motion/P_PID_antibacklash
(*This Program is built for antibacklash of azimuth and elevation,using PID function block*)
PROGRAM P_PID_antibacklash
VAR
(*<<<<<<<<<<<<<<<<<<azimuth>>>>>>>>>>>>*)
	FB_PID_AZ: IL_PIDType01;
	//DT_IControl_az:TIME:=T#50MS;
	DT_IControl_az:TIME:=T#20MS;(*The integration time Tn for the integration portion of the controller.*)
	r_PControl_az: REAL:=0.0001;(*The proportional value of the gain portion of the controller.*)
	r_Setpoint_az:REAL:=0;(*The desired "Setpoint" for the controlled process*)
	r_controlvalue_az: REAL;(*The calculated controller output value*)
	r_PID_feedback_az: REAL;(*The current actual value of the process*)
(*<<<<<<<<<<<<<<<<<<elevation>>>>>>>>>>>>*)
	FB_PID_EL: IL_PIDType01;
	DT_Icontrol_el:TIME;
	r_PControl_el: REAL;
(*r_Setpoint_el:REAL:=-40;*)(*only for Antenna #4*)
	r_Setpoint_el:REAL:=-5;
	r_controlvalue_el: REAL;
	r_PID_feedback_EL: REAL;
	
(*<<<<<<<<<<<<<<<<<<FeedIndexer>>>>>>>>>>>>*)
	FB_PID_FI: IL_PIDType01;
	DT_IControl_FI:TIME:=T#20MS;(*The integration time Tn for the integration portion of the controller.*)
	r_PControl_FI: REAL:=0.0001;(*The proportional value of the gain portion of the controller.*)
	r_Setpoint_FI:REAL:=-10;(*The desired "Setpoint" for the controlled process*)
	r_controlvalue_FI: REAL;(*The calculated controller output value*)
	r_PID_feedback_FI: REAL;(*The current actual value of the process*)	
	test1: BOOL;
	test3: BOOL;
	test4: BOOL;
	tre: BOOL;
END_VAR

P_PID_antibacklash.A_PID();
(***********************************change the bias when enable off**********************************)
IF b_off_write=TRUE THEN
	r_Setpoint_az:=10;
	r_Setpoint_el:=0;
	r_Setpoint_FI:=0;
ELSE
	r_Setpoint_az:=10;
	r_Setpoint_el:=-5;
	r_Setpoint_FI:=-5;
END_IF

(*<<<<<<<<<<<<<<<<<<<<<<<<<<<<<<<<<<<<<<<Azimuth>>>>>>>>>>>>>>>>>>>>>>>>>>>>>>>>>>>>>>>>>>>>>>>>*)
r_PID_feedback_az:=axisdata[2].rActualTorqueForce_i-axisdata[1].rActualTorqueForce_i;
IF b_PID_in_az=TRUE THEN
	axisdata[2].dwUserCmdDataB_q.REAL_:=r_controlvalue_az;
(*axisdata[2].rActualTorqueForce_i is set to the parameter P690,additional velocity value.*)
ELSE
	axisdata[2].dwUserCmdDataB_q.REAL_:=0;
END_IF;
(*<<<<<<<<<<<<<<<<<<<<<<<<<<<<<<<<<<<<<<<Elevation>>>>>>>>>>>>>>>>>>>>>>>>>>>>>>>>>>>>>>>>>>>>>>>>*)
r_PID_feedback_el:=axisdata[4].rActualTorqueForce_i-axisdata[3].rActualTorqueForce_i;
IF b_gearin_4_done=TRUE THEN
	axisdata[4].dwUserCmdDataB_q.REAL_:=r_controlvalue_el;
ELSE
	axisdata[4].dwUserCmdDataB_q.REAL_:=0;
END_IF;
(*<<<<<<<<<<<<<<<<<<<<<<<<<<<<<<<<<<<<<<<FeedIndexer>>>>>>>>>>>>>>>>>>>>>>>>>>>>>>>>>>>>>>>>>>>>>>>>*)
r_PID_feedback_FI:=axisdata[6].rActualTorqueForce_i-axisdata[5].rActualTorqueForce_i;
IF b_gearin_6_done=TRUE THEN
	axisdata[6].dwUserCmdDataB_q.REAL_:=r_controlvalue_FI;
ELSE
	axisdata[6].dwUserCmdDataB_q.REAL_:=0;
END_IF;

(*		DT_Icontrol_az:=T#20MS;
		r_PControl_az:=0.0001;
		DT_Icontrol_el:=T#20MS;
		r_PControl_el:=0.00008;
		DT_Icontrol_FI:=T#20MS;
		r_PControl_FI:=0.00005;
*)
(*
(****************************PID parameter*********************************)
str_1xx:=RIGHT(str_MLC_ip,3);(*get the IP address of MLC*)
IF r_pos_az>=358.5 OR r_pos_az<=-178.5 THEN
	DT_Icontrol_az:=T#40ms;
	r_PControl_az:=0.000001;
END_IF;

IF  r_pos_az<358.5 OR r_pos_az>-178.5 THEN
	IF str_1xx='188' OR  str_1xx='188' OR str_1xx='188' OR  str_1xx='188' THEN
		DT_Icontrol_az:=T#20ms;
		r_PControl_az:=0.00006;
	ELSE
		DT_Icontrol_az:=T#20ms;
		r_PControl_az:=0.0001;
	END_IF;
END_IF;



IF r_pos_el>=90.10 OR r_pos_el<=15.5 THEN
	DT_Icontrol_el:=T#40ms;
	r_PControl_el:=0.000001;
END_IF;

IF r_pos_el<90.10 AND r_pos_el>15.5 THEN
	IF str_1xx='188' OR  str_1xx='188' OR str_1xx='188' OR  str_1xx='188' THEN
		DT_Icontrol_el:=T#20ms;
		r_PControl_el:=0.00006;
	ELSE
		DT_Icontrol_el:=T#20ms;
		r_PControl_el:=0.00008;
	END_IF;
END_IF;
*)

ACTION A_PID:
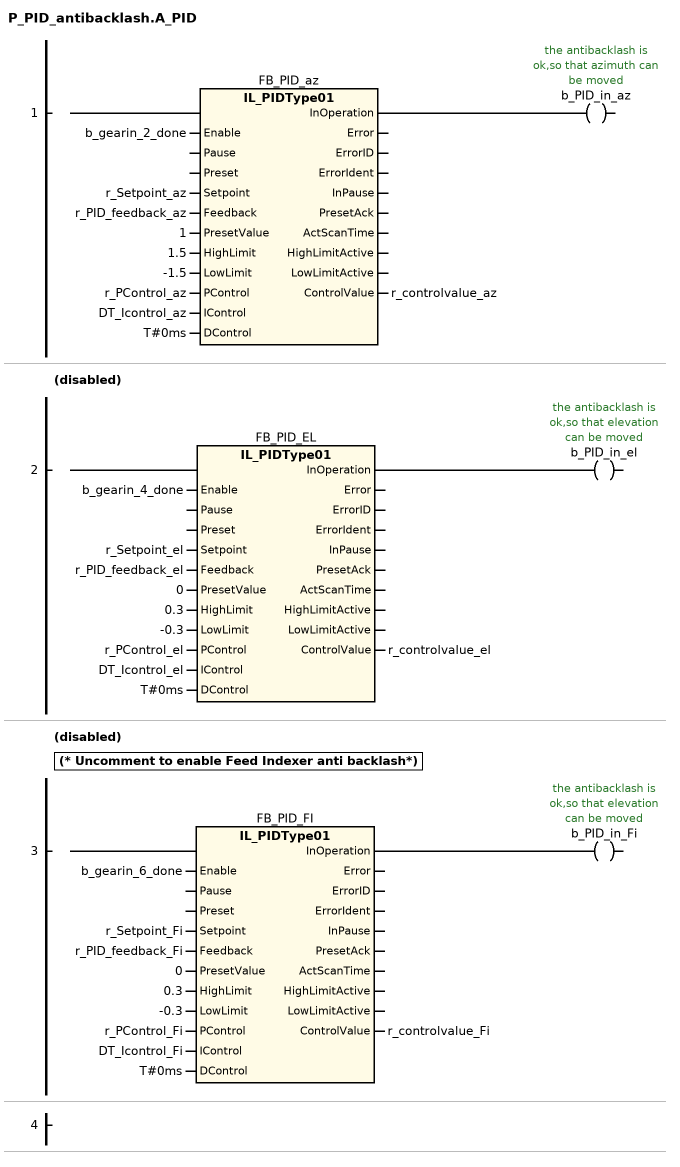
// NETWORK 1
//   FB_PID_az: <<<<<<<<<<<<<<<<<<azimuth>>>>>>>>>>>>
//   b_gearin_2_done: drive 1 and 2 are synchronous with v_azimuth
//   r_Setpoint_az: The desired "Setpoint" for the controlled process
//   r_PID_feedback_az: The current actual value of the process
//   r_PControl_az: The proportional value of the gain portion of the controller.
//   DT_Icontrol_az: The integration time Tn for the integration portion of the controller.
//   r_controlvalue_az: The calculated controller output value
//   b_PID_in_az: the antibacklash is ok,so that azimuth can be moved
FB_PID_az(
    Enable := b_gearin_2_done,
    Setpoint := r_Setpoint_az,
    Feedback := r_PID_feedback_az,
    PresetValue := 1,
    HighLimit := 1.5,
    LowLimit := -1.5,
    PControl := r_PControl_az,
    IControl := DT_Icontrol_az,
    DControl := T#0ms,
    ControlValue => r_controlvalue_az); // IL_PIDType01
b_PID_in_az := FB_PID_az.InOperation;

// NETWORK 2 (disabled)
//   FB_PID_EL: <<<<<<<<<<<<<<<<<<elevation>>>>>>>>>>>>
//   b_gearin_4_done: drive 3 and 4 are synchronous with v_elevation
//   r_Setpoint_el: r_Setpoint_el:REAL:=-40; only for Antenna #4
//   b_PID_in_el: the antibacklash is ok,so that elevation can be moved
// FB_PID_EL(
//     Enable := b_gearin_4_done,
//     Setpoint := r_Setpoint_el,
//     Feedback := r_PID_feedback_el,
//     PresetValue := 0,
//     HighLimit := 0.3,
//     LowLimit := -0.3,
//     PControl := r_PControl_el,
//     IControl := DT_Icontrol_el,
//     DControl := T#0ms,
//     ControlValue => r_controlvalue_el); // IL_PIDType01
// b_PID_in_el := FB_PID_EL.InOperation;

// NETWORK 3 (disabled)
//   FB_PID_FI: <<<<<<<<<<<<<<<<<<elevation>>>>>>>>>>>>
//   b_gearin_6_done: drive 3 and 4 are synchronous with v_elevation
//   r_Setpoint_Fi: r_Setpoint_el:REAL:=-40; only for Antenna #4
//   b_PID_in_Fi: the antibacklash is ok,so that elevation can be moved
// label: (* Uncomment to enable Feed Indexer anti backlash*)
// FB_PID_FI(
//     Enable := b_gearin_6_done,
//     Setpoint := r_Setpoint_Fi,
//     Feedback := r_PID_feedback_Fi,
//     PresetValue := 0,
//     HighLimit := 0.3,
//     LowLimit := -0.3,
//     PControl := r_PControl_Fi,
//     IControl := DT_Icontrol_Fi,
//     DControl := T#0ms,
//     ControlValue => r_controlvalue_Fi); // IL_PIDType01
// b_PID_in_Fi := FB_PID_FI.InOperation;

// NETWORK 4
END_ACTION

END_PROGRAM

// IndraMotionMlc1/Application/POUs/Time Control/P_UDP_To_NTP
(*This program is built for use the NTP protocol to update the time by using
the UDP package, then update the MLC time*)
PROGRAM P_UDP_To_NTP
VAR
(*UDP function block*)
	FB_UDP_Async_Start: IL_UDPSocketAsync;
	strIP_adress:ARRAY [1..3] OF STRING;
	strIP: STRING:='192.168.1.5';
	Int_adress: INT := 1;
	uiport:UINT:=123;
	UDP_bConnectionEstablished: BOOL;
	UDP_Server_Enable: BOOL;
	UDP_diSocket: DINT;
	FB_UDP_Send: IL_UDPSendtoAsync;
	UDP_bRecv: BOOL;
	diSentBytes: DINT;
	FB_UDP_Receive: IL_UDPRecvfromAsync;
	UDP_bSent: BOOL;
	UDP_bSend: BOOL;
	UDP_bReceived: BOOL;
	UDP_diReceivedBytes: UDINT;
(*NTP define*)
	st_UDP_SendPacket:UDP_PACKET;(*packet of send*)
	st_UDP_ReceivePacket:UDP_PACKET;(*packet of recieve*)
(*NTP header definition *)
	S_LeapYearIndicator: BYTE;(*2bit*)
	S_VersionNumber: BYTE;(*3bit*)
	S_Stratum : BYTE;(*8bit*)
	S_Mode : BYTE;(*3bit*)
	S_FIlInterval : BYTE;(*8bit*)
	S_Percision : BYTE;(*8bit*)
	S_Root_delay : DWORD;(*32bit*)
	S_Root_Dispersion : DWORD;(*32bit*)
	S_Reference_Identifier: DWORD;(*32bit*)
(*4 time stamps*)
	S_Reference_Timestamp:ARRAY[1..2] OF DWORD;
	S_Originate_Timestamp:ARRAY[1..2] OF DWORD;
	S_Receive_Timestamp:ARRAY[1..2] OF DWORD;
	S_Transmit_Timestamp:ARRAY[1..2] OF DWORD;
(*convert MJD to UTC*)
    Dwordtime_second:DWORD;
    Dwordtime_Millisecond:DWORD;
(*4 time stamps of NTP need*)
    T1:LREAL;
	T2:LREAL;
	T3:LREAL;
	T4:LREAL;
	UTCcurrenttime:LREAL;
	SysTimeNTP: DT;
(*convert the updated time stamps to UTC*)
    UTC_to_MJD_day:REAL;
    UTC_to_MJD_second:LREAL;
	mjd_UTCtime_day:REAL;
	mjd_UTCtime_second:LREAL;
	mjd_UTCtime_Millisecond:LREAL;
(*translate the order between the big endian and small endian*)
	org_to_net_high:IL_DWordToByte;
    org_to_net_low:IL_DWordToByte;
    org_time_high:DWORD;
    org_time_low:DWORD;
    org_nettime_high:DWORD;
    org_nettime_low:DWORD;
	rev_to_local_high:IL_DWordToByte;
    rev_to_local_low:IL_DWordToByte;
    rev_nettime_high:DWORD;
    rev_nettime_low:DWORD;
    rev_time_high:DWORD;
    rev_time_low:DWORD;
	tran_to_local_high:IL_DWordToByte;
    tran_to_local_low:IL_DWordToByte;
    tran_nettime_high:DWORD;
    tran_nettime_low:DWORD;
    tran_time_high:DWORD;
    tran_time_low:DWORD;
(*<<<<<<<<<<<<<<<<<<<<<<<<<<<<<>>>>>>>>>>>>>>>>>>>>>>>>>>>>>>>>>>>>>>>>*)
	
	fb_rtri_start: R_TRIG;
	fb_rtri_receive_end: R_TRIG;
	FB_RESET_UDP: R_TRIG;
	fb_error_reset: TON;
	b_mjd_need_updata: BOOL;
	ton_updata_need: TON;
	rtrig_need: R_TRIG;
	FB_M_time_move: MC_MoveAbsolute;
	FB_clear_all_error: MB_WriteParameter;
	b_clear_done: BOOL;
	
	FB_Time_master: MC_MoveVelocity;
	fb_stop_v_time: MC_Stop;
	b_stop_v_time_done: BOOL;
	rtrig_reset_all: R_TRIG;
	detaT:LREAL;
	b_server: BOOL:=FALSE;
	i_hour: INT;
	b_update_hour_NTP: BOOL;
	fb_r_trig_updata_NTP:R_TRIG;
	fb_r_trig_reset_ntp: R_TRIG;
	i_NTP_count: INT;
	ton_ntp_timeout: TON;
	b_ntp_timeout: BOOL;
	fftrig_track_off: F_TRIG;
	test_second:LREAL;
	test_second1:LREAL;
	test_second2:LREAL;
	test_second4:LREAL;
	test_second3:UDINT;
	r_time_speed: LREAL;
	IL_SetDateTime_0: IL_SetDateTime;
	SysTimeUpdate: DATE_AND_TIME;
	b_sys_time_done: BOOL;
	test: BOOL;
END_VAR

VAR_INPUT 
	b_NTP_set_up:BOOL;
	current_time_pos:LREAL;
END_VAR

r_time_speed:=1.0/6.0;

//r_time_speed:=0.1666666666667;
IF Time_cds.Status.DscTimeSyncSource = 1 THEN
(*update the time when the system already started*)
strIP_adress[1] := Time_cds.Status.TimeSourceAddrNTP;
strIP_adress[2] := Time_cds.Status.TimeSourceAddrNTP;
strIP_adress[3] := Time_cds.Status.TimeSourceAddrNTP;
IF b_NTP_set_up = TRUE THEN
	Int_adress:=1;
	strIP:=Time_cds.Status.TimeSourceAddrNTP;;
END_IF;

WHILE b_ntp_timeout = TRUE DO
Int_adress := Int_adress+1;
 IF Int_adress>3 THEN
	Int_adress:=1;
 END_IF;
strIP:= strIP_adress[Int_adress];
b_ntp_update_start:= FALSE;
b_ntp_timeout := FALSE;
END_WHILE;

IF di_MJD_day<10000 AND b_NTP_update_start=FALSE AND axisdata[1].Axis_Inbb THEN
	b_mjd_need_updata:=TRUE;
ELSE
	b_mjd_need_updata:=FALSE;
END_IF

(*update the time every 15 mins*)
FOR i_hour := 0 TO 23 BY 1 DO
	IF i_num_quarter=i_hour*4+1 THEN
		b_update_hour_NTP:=TRUE;
	ELSE
		b_update_hour_NTP:=FALSE;
	END_IF;
END_FOR;

(*the update action is springed by the raise edge*)
fb_r_trig_updata_NTP(clk:=b_update_hour_NTP);
IF fb_r_trig_updata_NTP.Q = TRUE THEN
	b_ntp_update_start:=TRUE;
END_IF;
(*when the update start,spring a raise edge to send and receive UDP package *)
fb_rtri_start(clk:=b_NTP_update_start);
fb_rtri_receive_end(clk:=UDP_bReceived);
IF fb_rtri_start.Q =TRUE THEN
(*<<<<<<<<<<<<<<<<<<<<<<<<<<<<value the send packet>>>>>>>>>>>>>>>>>>>>>>>>>>>>>>>>>>>>>>>>>>>>>*)
	S_LeapYearIndicator.0:=0;
	S_LeapYearIndicator.1:=0;
	S_VersionNumber.0:=1;
	S_VersionNumber.1:=1;
	S_VersionNumber.2:=0;
	S_Mode.0:=1;
	S_Mode.1:=1;
	S_Mode.2:=0;
	S_Stratum:=0;
	S_FIlInterval:=0;
	S_Percision:=0;
	S_Root_Dispersion:=0;
	S_Reference_Identifier:=0;
(*<<<<<<<<<<<<<<<<<<<<<<<<<<<<<<<<<<calculate the time stamps>>>>>>>>>>>>>>>>>>>>>>>>>>>>>>>*)
	UDP_Server_Enable:=TRUE;
	mjd_UTCtime_day:=TRUNC(lr_MJD_current)-40587;
mjd_UTCtime_second:=mjd_UTCtime_day*86400+2208988800+TRUNC((lr_MJD_current-TRUNC(lr_MJD_current))*86400)+128;
mjd_UTCtime_Millisecond:=(lr_MJD_current-TRUNC(lr_MJD_current))*86400-TRUNC((lr_MJD_current-TRUNC(lr_MJD_current))*86400);
(*<<<<<<<<<<<<<<<<<<<<<<<<<<<<<<<<<<<<<<<<<<<<value the head og send packet>>>>>>>>>>>>>>>>>>>>>>>>>>>>>>>>>>>>>>>>>>>>>>>>>>>*)
	st_UDP_SendPacket.NTP_Header:=F_NTP_Head(S_LeapYearIndicator,S_VersionNumber,S_Stratum,S_Mode,S_FIlInterval,S_Percision);
	st_UDP_SendPacket.NTP_Root_Delay[1]:=0;
	st_UDP_SendPacket.NTP_Root_Delay[2]:=0;
	st_UDP_SendPacket.NTP_Root_Delay[3]:=0;
	st_UDP_SendPacket.NTP_Root_Delay[4]:=0;
	st_UDP_SendPacket.NTP_Root_Dispersion[1]:=0;
	st_UDP_SendPacket.NTP_Root_Dispersion[2]:=0;
	st_UDP_SendPacket.NTP_Root_Dispersion[3]:=0;
	st_UDP_SendPacket.NTP_Root_Dispersion[4]:=0;
	st_UDP_SendPacket.NTP_Reference_Identifier[1]:=0;
	st_UDP_SendPacket.NTP_Reference_Identifier[2]:=0;
	st_UDP_SendPacket.NTP_Reference_Identifier[3]:=0;
	st_UDP_SendPacket.NTP_Reference_Identifier[4]:=0;

	org_time_high:=LREAL_TO_DWORD(mjd_UTCtime_second);
	org_time_low:=LREAL_TO_DWORD(mjd_UTCtime_Millisecond*1000);
	(*originate Timestamp to net word*)
	org_to_net_high(Input:=org_time_high);
	org_nettime_high:=IL_ByteToDWord(org_to_net_high.Byte3,org_to_net_high.Byte2,org_to_net_high.Byte1,org_to_net_high.Byte0);

	org_to_net_low(Input:=org_time_low);
	org_nettime_low:=IL_ByteToDWord(org_to_net_low.Byte3,org_to_net_low.Byte2,org_to_net_low.Byte1,org_to_net_low.Byte0);

	st_UDP_SendPacket.NTP_Reference_Timestamp[1]:=0;
	st_UDP_SendPacket.NTP_Reference_Timestamp[2]:=0;
	st_UDP_SendPacket.NTP_Originate_Timestamp[1]:=0;
	st_UDP_SendPacket.NTP_Originate_Timestamp[2]:=0;
	st_UDP_SendPacket.NTP_Receive_Timestamp[1]:=0;
	st_UDP_SendPacket.NTP_Receive_Timestamp[2]:=0;
	st_UDP_SendPacket.NTP_Transmit_Timestamp[1]:=org_nettime_high;
	st_UDP_SendPacket.NTP_Transmit_Timestamp[2]:=org_nettime_low;
	UDP_bSend:=TRUE;
	UDP_bRecv:=TRUE;
END_IF;
(*at the same time, open the receive channels*)
IF fb_rtri_receive_end.Q =TRUE THEN
(*recalculate the current time*)
	mjd_UTCtime_day:=TRUNC(lr_MJD_current)-40587;
	mjd_UTCtime_second:=mjd_UTCtime_day*86400+2208988800+TRUNC((lr_MJD_current-TRUNC(lr_MJD_current))*86400)+128;
	mjd_UTCtime_Millisecond:=(lr_MJD_current-TRUNC(lr_MJD_current))*86400-TRUNC((lr_MJD_current-TRUNC(lr_MJD_current))*86400);
	Dwordtime_second:=LREAL_TO_DWORD(mjd_UTCtime_second);
    Dwordtime_Millisecond:=LREAL_TO_DWORD(mjd_UTCtime_Millisecond*1000);
	rev_nettime_high:=st_UDP_ReceivePacket.NTP_Receive_Timestamp[1];
	rev_nettime_low:=st_UDP_ReceivePacket.NTP_Receive_Timestamp[2];
	tran_nettime_high:=st_UDP_ReceivePacket.NTP_Transmit_Timestamp[1];
	tran_nettime_low:=st_UDP_ReceivePacket.NTP_Transmit_Timestamp[2];
(*translate the big endian to small endian*)
	rev_to_local_high(Input:=rev_nettime_high);
	rev_time_high:=IL_ByteToDWord(rev_to_local_high.Byte3,rev_to_local_high.Byte2,rev_to_local_high.Byte1,rev_to_local_high.Byte0);
	rev_to_local_low(Input:=rev_nettime_low);
	rev_time_low:=IL_ByteToDWord(rev_to_local_low.Byte3,rev_to_local_low.Byte2,rev_to_local_low.Byte1,rev_to_local_low.Byte0);
	tran_to_local_high(Input:=tran_nettime_high);
	tran_time_high:=IL_ByteToDWord(tran_to_local_high.Byte3,tran_to_local_high.Byte2,tran_to_local_high.Byte1,tran_to_local_high.Byte0);
	tran_to_local_low(Input:=tran_nettime_low);
	tran_time_low:=IL_ByteToDWord(tran_to_local_low.Byte3,tran_to_local_low.Byte2,tran_to_local_low.Byte1,tran_to_local_low.Byte0);
(*calculate the four timestamp for calculating the right time*)
	T1:=DWORD_TO_LREAL(org_time_high)+DWORD_TO_LREAL(org_time_low)/1000;
	T2:=DWORD_TO_LREAL(rev_time_high)+DWORD_TO_LREAL(rev_time_low)/4294967296;
	T3:=DWORD_TO_LREAL(tran_time_high)+DWORD_TO_LREAL(tran_time_low)/4294967296;
	T4:=DWORD_TO_LREAL(Dwordtime_second)+DWORD_TO_LREAL(Dwordtime_Millisecond)/1000;
(*the difference time is detaT*)
	detaT:=(T2-T1)/2-(T4-T3)/2;
(*the update time is T4+detaT, the 0.015 is the delay of running time*)
	UTCcurrenttime:=T4+detaT-0.015;
(*calculate the MJD day and MJD second*)
	UTC_to_MJD_day:=TRUNC(UTCcurrenttime-2208988800)/86400+40587;
	test_second2:=UTCcurrenttime/86400;
	test_second3:=TRUNC(test_second2);
	test_second4:=UDINT_TO_LREAL(test_second3*86400);
	test_second1:=TRUNC(UTCcurrenttime/86400)*86400;
	UTC_to_MJD_second:=UTCcurrenttime-UDINT_TO_LREAL(TRUNC(UTCcurrenttime/86400)*86400);
(*<<<<<<<<<<<<<<<<<<<<<<<<<<<<<<<<<<<not update untill track off>>>>>>>>>>>>>>>>>>>>>>>>>>>>>>>>>>>>>>>>*)
	IF b_track_on=FALSE  THEN
(*prohibit the update process when the system is tracking,otherwise it will bring the time jump and disturb the trajectory*)
		di_MJD_day:=REAL_TO_DINT(UTC_to_MJD_day);
		i_num_quarter:=TRUNC(UTC_to_MJD_second/360);
		test_second:=i_num_quarter*360;
		current_time_pos:=UTC_to_MJD_second-i_num_quarter*360;(*the needed position of time master axis*)
		i_NTP_count:=i_NTP_count+1;
		b_NTP_set_up:=TRUE;
		detaT:=0;
	END_IF;
(*if the difference time>0.08, then update time *)
END_IF;

IF ABS(detaT)>0.08 THEN
		B_NTP_NEED_UPDATE:=TRUE;
ELSE
		B_NTP_NEED_UPDATE:=FALSE;
END_IF

END_IF
(*transfer the sub-program for communicating and update time*)
SysTimeUpdate:=LREAL_TO_DT(UTCcurrenttime-2208988800);
P_UDP_To_NTP.A_UDP();
P_UDP_To_NTP.A_NTP_to_Master();

ACTION A_NTP_to_Master:
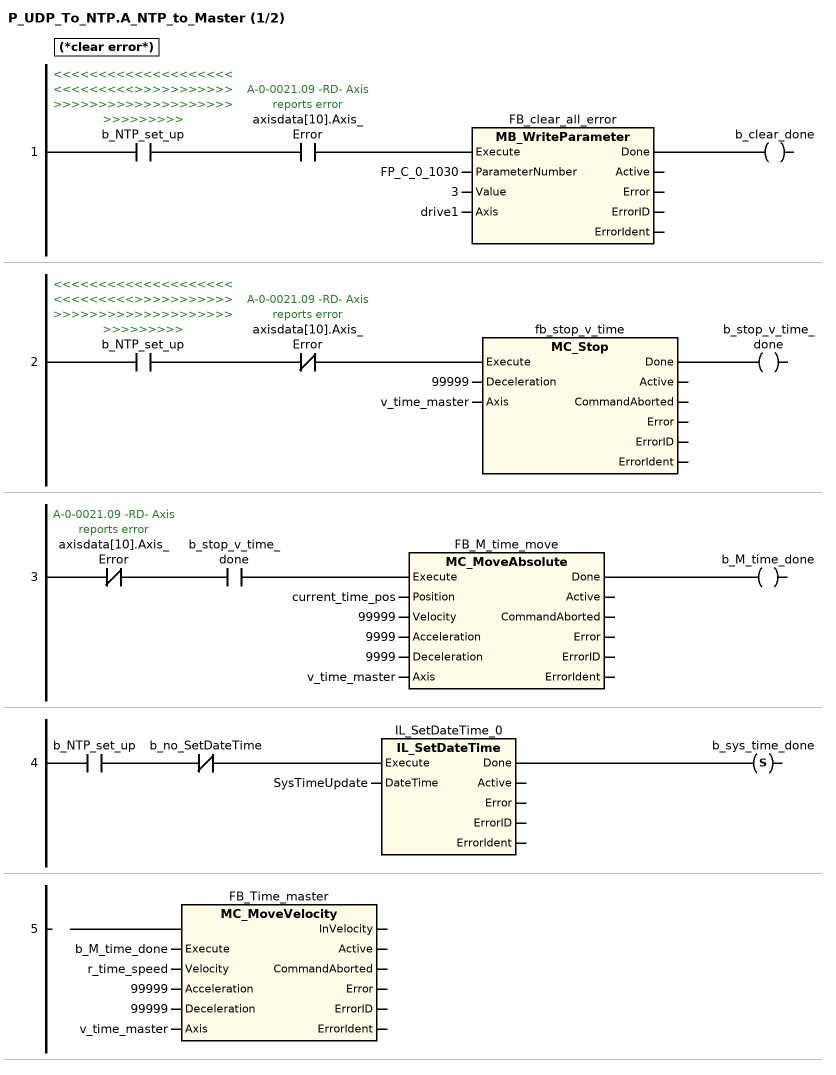
// NETWORK 1
//   b_NTP_set_up: <<<<<<<<<<<<<<<<<<<<<<<<<<<<<>>>>>>>>>>>>>>>>>>>>>>>>>>>>>>>>>>>>>>>>
//   axisdata[10].Axis_Error: A-0-0021.09 -RD- Axis reports error
//   FP_C_0_1030: Command: Clear all control errors
//   drive1: Real axis "Drive1" with axis number 1
// label: (*clear error*)
FB_clear_all_error(
    Execute := b_NTP_set_up AND axisdata[10].Axis_Error,
    ParameterNumber := FP_C_0_1030,
    Value := 3,
    Axis := drive1); // MB_WriteParameter
b_clear_done := FB_clear_all_error.Done;

// NETWORK 2
//   b_NTP_set_up: <<<<<<<<<<<<<<<<<<<<<<<<<<<<<>>>>>>>>>>>>>>>>>>>>>>>>>>>>>>>>>>>>>>>>
//   axisdata[10].Axis_Error: A-0-0021.09 -RD- Axis reports error
//   v_time_master: Virtual axis "v_time_master" with axis number 10
fb_stop_v_time(
    Execute := b_NTP_set_up AND NOT axisdata[10].Axis_Error,
    Deceleration := 99999,
    Axis := v_time_master); // MC_Stop
b_stop_v_time_done := fb_stop_v_time.Done;

// NETWORK 3
//   axisdata[10].Axis_Error: A-0-0021.09 -RD- Axis reports error
//   v_time_master: Virtual axis "v_time_master" with axis number 10
FB_M_time_move(
    Execute := NOT axisdata[10].Axis_Error AND b_stop_v_time_done,
    Position := current_time_pos,
    Velocity := 99999,
    Acceleration := 9999,
    Deceleration := 9999,
    Axis := v_time_master); // MC_MoveAbsolute
b_M_time_done := FB_M_time_move.Done;

// NETWORK 4
IL_SetDateTime_0(Execute := b_NTP_set_up AND NOT b_no_SetDateTime, DateTime := SysTimeUpdate); // IL_SetDateTime
b_sys_time_done S= IL_SetDateTime_0.Done;

// NETWORK 5
//   v_time_master: Virtual axis "v_time_master" with axis number 10
FB_Time_master(
    Execute := b_M_time_done,
    Velocity := r_time_speed,
    Acceleration := 99999,
    Deceleration := 99999,
    Axis := v_time_master); // MC_MoveVelocity

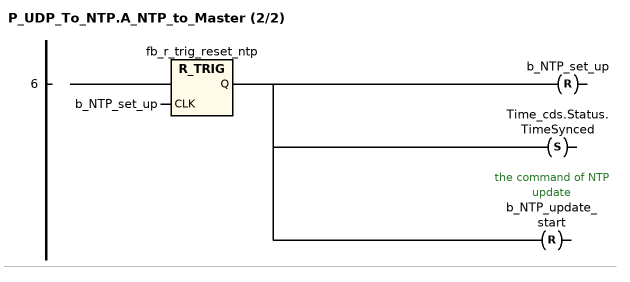
// NETWORK 6
//   b_NTP_set_up: <<<<<<<<<<<<<<<<<<<<<<<<<<<<<>>>>>>>>>>>>>>>>>>>>>>>>>>>>>>>>>>>>>>>>
//   b_NTP_update_start: the command of NTP update
fb_r_trig_reset_ntp(CLK := b_NTP_set_up); // R_TRIG
b_NTP_set_up R= fb_r_trig_reset_ntp.Q;
Time_cds.Status.TimeSynced S= fb_r_trig_reset_ntp.Q;
b_NTP_update_start R= fb_r_trig_reset_ntp.Q;
END_ACTION

ACTION A_UDP:
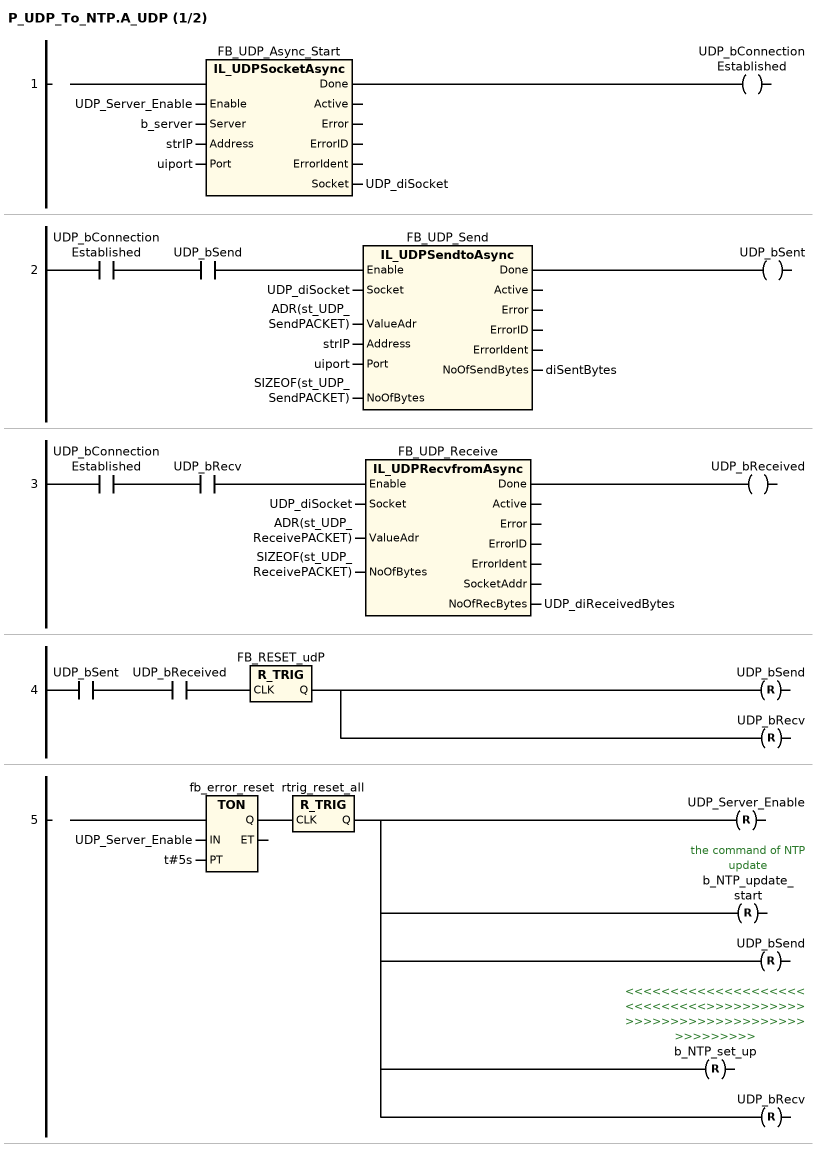
// NETWORK 1
//   FB_UDP_Async_Start: UDP function block
FB_UDP_Async_Start(
    Enable := UDP_Server_Enable,
    Server := b_server,
    Address := strIP,
    Port := uiport,
    Socket => UDP_diSocket); // IL_UDPSocketAsync
UDP_bConnectionEstablished := FB_UDP_Async_Start.Done;

// NETWORK 2
FB_UDP_Send(
    Enable := UDP_bConnectionEstablished AND UDP_bSend,
    Socket := UDP_diSocket,
    ValueAdr := ADR(st_UDP_SendPACKET),
    Address := strIP,
    Port := uiport,
    NoOfBytes := SIZEOF(st_UDP_SendPACKET),
    NoOfSendBytes => diSentBytes); // IL_UDPSendtoAsync
UDP_bSent := FB_UDP_Send.Done;

// NETWORK 3
FB_UDP_Receive(
    Enable := UDP_bConnectionEstablished AND UDP_bRecv,
    Socket := UDP_diSocket,
    ValueAdr := ADR(st_UDP_ReceivePACKET),
    NoOfBytes := SIZEOF(st_UDP_ReceivePACKET),
    NoOfRecBytes => UDP_diReceivedBytes); // IL_UDPRecvfromAsync
UDP_bReceived := FB_UDP_Receive.Done;

// NETWORK 4
FB_RESET_udP(CLK := UDP_bSent AND UDP_bReceived); // R_TRIG
UDP_bSend R= FB_RESET_udP.Q;
UDP_bRecv R= FB_RESET_udP.Q;

// NETWORK 5
//   b_NTP_update_start: the command of NTP update
//   b_NTP_set_up: <<<<<<<<<<<<<<<<<<<<<<<<<<<<<>>>>>>>>>>>>>>>>>>>>>>>>>>>>>>>>>>>>>>>>
fb_error_reset(IN := UDP_Server_Enable, PT := t#5s); // TON
rtrig_reset_all(CLK := fb_error_reset.Q); // R_TRIG
UDP_Server_Enable R= rtrig_reset_all.Q;
b_NTP_update_start R= rtrig_reset_all.Q;
UDP_bSend R= rtrig_reset_all.Q;
b_NTP_set_up R= rtrig_reset_all.Q;
UDP_bRecv R= rtrig_reset_all.Q;

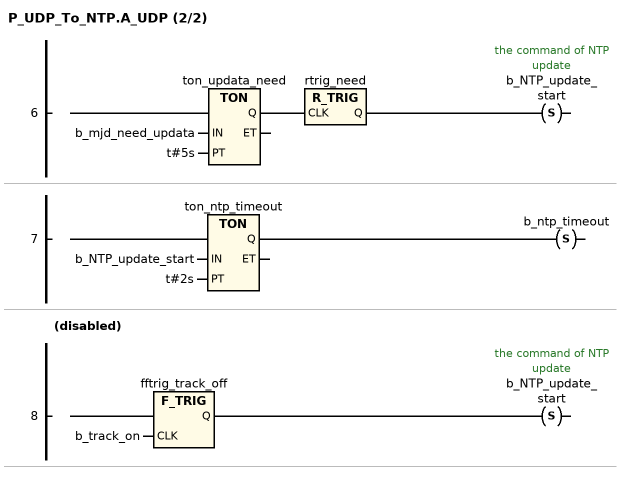
// NETWORK 6
//   b_NTP_update_start: the command of NTP update
ton_updata_need(IN := b_mjd_need_updata, PT := t#5s); // TON
rtrig_need(CLK := ton_updata_need.Q); // R_TRIG
b_NTP_update_start S= rtrig_need.Q;

// NETWORK 7
//   b_NTP_update_start: the command of NTP update
ton_ntp_timeout(IN := b_NTP_update_start, PT := t#2s); // TON
b_ntp_timeout S= ton_ntp_timeout.Q;

// NETWORK 8 (disabled)
//   b_track_on: the command of running trajectory
//   b_NTP_update_start: the command of NTP update
// fftrig_track_off(CLK := b_track_on); // F_TRIG
// b_NTP_update_start S= fftrig_track_off.Q;
END_ACTION

END_PROGRAM

// IndraMotionMlc1/Application/POUs/Time Control/F_NTP_Head
(*This program is built for establishing a model that according to the standard of UDP package*)
(*<<<<<<<<<<<<<<<<<<<<NTP head,16byte>>>>>>>>>>>>>>>>>>>>>>>*)
FUNCTION F_NTP_Head : ARRAY [1..4] OF BYTE
VAR_INPUT
	LeapYearIndicator: BYTE;(*2bit*)
	VersionNumber: BYTE;(*3bit*)
	Stratum : BYTE;(*8bit*)
	Mode : BYTE;(*3bit*)
	FIlInterval : BYTE;(*8bit*)
	Percision : BYTE;(*8bit*)
END_VAR
VAR
(*<<<<<<<<<<<<<<<<<<<DWORD to BYTE>>>>>>>>>>>>>>>>>>>>>>>*)
	dword_to_byte_R_I:IL_DWordToByte;
	dword_to_byte_R_Dis:IL_DWordToByte;
	dword_to_byte_R_Delay:IL_DWordToByte;
	dword_to_byte_R_D: BOOL;
END_VAR

(*Percision value*)
F_NTP_Head[4]:=Percision;
(*FIlInterval vlue*)
F_NTP_Head[3]:=FIlInterval;
(*LeapYearIndicator VersionNumber Stratum Mode*)
F_NTP_Head[2]:=IL_BoolToByte(stratum.0,stratum.1,stratum.2,stratum.3,stratum.4,stratum.5,stratum.6,stratum.7);
F_NTP_Head[1]:=IL_BoolToByte(mode.0,mode.1,mode.2,VersionNumber.0,VersionNumber.1,VersionNumber.2,LeapYearIndicator.0,LeapYearIndicator.1);

END_FUNCTION

// IndraMotionMlc1/Application/POUs/Motion/POU_20200525
PROGRAM POU_20200525
VAR
	MB_ReadParameter_P434: MB_ReadrealParameter;
	Cyclic_position: LREAL;
	Cal_followingError: LREAL;
	delta_E:LREAL;
	delta_E_modify:LREAL;
END_VAR

(*arAxisStatus_gb[3].AxisData_HMI.Axis_InSynchron;
arAxisStatus_gb[3].Admin._OpModeAck;
ML_Base.AxisData[3].Axis_Power;
(*
MB_ReadParameter_P434(
	Enable:= TRUE, 
	Done=> , 
	Active=> , 
	Error=> , 
	ErrorID=> , 
	ErrorIdent=> , 
	ParameterNumber:=FP_P_0_0434 , 
	Value=> Cyclic_position, 
	Axis:= Drive3);
*)
Cal_followingError:=Cyclic_position-axisdata[3].rActualPosition_i;

delta_E:=r_write_position_el-axisdata[3].rActualPosition_i;
delta_E_modify:=r_write_position_el-P_Track_cubic.V0_el/86400-axisdata[3].rActualPosition_i;
//delta_E_modify:=Cyclic_position-axisdata[3].rActualPosition_i-axisdata[3].rActualVelocity_i;
//RATIO_INPUT := DINT_TO_UINT(TRUNC(gear_ratio*20));
//RATIO_OUTPUT := 26000;

IF P_power_on_TCP.b_M_el_done  THEN
(*	arAxisCtrl_gb[Drive3.AxisNo].SyncMode.Master := v_elevation;
	arAxisCtrl_gb[Drive3.AxisNo].SyncMode.StartMode := MC_START_MODE.ABSOLUTE_RAMPIN;
	arAxisCtrl_gb[Drive3.AxisNo].SyncMode.SyncDirection := MC_SYNC_DIRECTION.SHORTEST_WAY;
	arAxisCtrl_gb[Drive3.AxisNo].SyncMode.OutputRevolution := RATIO_INPUT;
	arAxisCtrl_gb[Drive3.AxisNo].SyncMode.InputRevolution := RATIO_OUTPUT;
	arAxisCtrl_gb[Drive3.AxisNo].SyncMode.SyncVelocity := 0.3;
	arAxisCtrl_gb[Drive3.AxisNo].SyncMode.SyncAcceleration := 0.03;*)
	//arAxisCtrl_gb[Drive3.AxisNo].Admin._OpMode.en := TechInterface.ModeAH;	
b_gearin_3_done:=TRUE;
END_IF


IF P_power_on_TCP.TEST2 OR b_SCC_enable_off THEN 
		arAxisCtrl_gb[Drive3.AxisNo].Admin._OpMode.en := Modeab;
END_IF

*)

END_PROGRAM

// IndraMotionMlc1/Application/POUs/Motion/P_Track_cubic
(*This program is built for running trajectory,and the trajectory runs by the rule y=ax^2+bx+c.
In this PROGRAM,there are two kinds OF FUNCTION blocks,ML_WriteCyclicPosition AND ML_OpenCyclicPositionChannel.
They are used for give the position command value to the virtual axis.*)
PROGRAM P_Track_cubic
VAR
(*azimuth,elevation and FeedIndexer position at i_start point *)
	p1_az: LREAL;
	p1_el: LREAL;
	p1_FI: LREAL;
(*azimuth,elevation and FeedIndexer position at i_start+1 point*)
	p2_az: LREAL;
	p2_el: LREAL;
	p2_FI: LREAL;
(*azimuth,elevation and FeedIndexer position at i_start+2 point*)
	p3_az: LREAL;
	p3_el: LREAL;
	p3_FI: LREAL;
(*the facters of the formula y=ax^2+bx+c*)
	a_az: LREAL;
	b_az: LREAL;
	a_el: LREAL;
	b_el: LREAL;
	a_FI: LREAL;
	b_FI: LREAL;
	t: LREAL;
	t1: LREAL;(*the time at i_start point*)
	t2: LREAL;(*the time at i_start+1 point*)
	t3: LREAL;(*the time at i_start+2 point*)
	
(*<<<<<<<<<<<<<<<<<<<<<<<<Write a Position value to azimuth,elevation and FeedIndexer virtual axis>>>>>>>>>>>>>>>>>>*)
	fb_write_positon_az: ML_WriteCyclicPosition;
	fb_write_positon_el: ML_WriteCyclicPosition;
	fb_write_positon_FI: ML_WriteCyclicPosition;

(*Open Cyclic Position Channel for azimuth,elevation and FeedIndexer.
Only if the cyclic position target value channel is open, 
the position command will become effective in the next cycle on the axis.*)
	fb_open_channel_az: ML_OpenCyclicPositionChannel;
	fb_open_channel_el: ML_OpenCyclicPositionChannel;
	fb_open_channel_FI: ML_OpenCyclicPositionChannel;

(*<<<<<<<<<<<<<definition for rtrig>>>>>>>>>>>>>>*)
	rtrig_track_on: R_TRIG;
	rtrig_write_position: R_TRIG;
	rtrig_reset_open_channel: R_TRIG;
	rtrig_reset_goto_track: R_TRIG;
	r_rtrig_start_stop:R_TRIG;
	ton_track_on:TON;
	b_signal_for_open: BOOL;
(*<<<<<<<<<<<<<<<<<<<<<<<the current position>>>>>>>>>>>>>>>>>>>*)
	r_last_position_az: LREAL;
	r_last_position_el: LREAL;
	r_last_position_FI: LREAL;
(*<<<<<<<<<<<<<<<<<<<<<<<<<<the current speed>>>>>>>>>>>>>>>>>>>>*)
	r_vel_last_az: LREAL;
	r_vel_last_el: LREAL;
	r_vel_last_FI: LREAL;
(*the distance and time between the current point and the first point*)
	r_start_distance_az: LREAL;
	r_start_distance_el: LREAL;
	r_start_distance_FI: LREAL;
	r_time_distance: LREAL;
(*the current velocity *)
	r_vel_start_az: LREAL;
	r_vel_start_el: LREAL;
	r_vel_start_FI: LREAL;
(*the transition for the azimuth position,r_write_position_az.*)
	r_calc_pos_az:LREAL;
	V0_el: LREAL;
	V0_az: LREAL;
	V0_FI: LREAL;
	i_point_caught: INT:=1;
	V_start_az: LREAL;
	V_start_el: LREAL;
	V_start_FI: LREAL;
	i_caught_MJD1:LREAL;
	i_caught_MJD2:LREAL;
	i_caught_TAIoffset1:LREAL;
	i_caught_TAIoffset2:LREAL;
	b_test:BOOL;
	
	i_start_first:INT;
	i_end_first:INT;
	
	test_1:INT;
	test_2:INT;
	
	r_start_az:LREAL;
	r_caught_az:LREAL;
	
	ton_pause_on:TON;
	rtrig_pause_on:R_TRIG;
	r_abs_az_speed:LREAL;
	r_abs_el_speed:LREAL;
	test_enable_el: BOOL;
	b_start_to_compensate: BOOL;
	p_covert_velocity:LREAL;
	r_following_test: LREAL;
	r_following_31: LREAL;
	r_following_333: LREAL;
	p_covert_velocity_el: LREAL;	
	(**********offset************)
	r_az_offset_Vmax:LREAL:=2.0;
	r_el_offset_Vmax:LREAL:=0.85;
	r_az_offset_acc:LREAL:=1.0;
	r_el_offset_acc:LREAL:=0.25;
	r_az_offset_dec:LREAL:=0.5;
	r_el_offset_dec:LREAL:=0.25;
	r_old_offset_az:LREAL;
	r_old_offset_el:LREAL;
	r_new_offset_az:LREAL;
	r_new_offset_el:LREAL;

	r_test_offset_az_abs:LREAL;
	r_test_offset_el_abs:LREAL;
	i_test_offset_count:DINT:=0;
	r_offset_t1_acc:LREAL;
	r_offset_t2_v:LREAL;
	r_offset_t3_dec:LREAL;
	l_offset_t1_acc:LREAL;
	l_offset_t2_v:LREAL;
	l_offset_t3_dec:LREAL;
	r_offset_t1_acc_el:LREAL;
	r_offset_t2_v_el:LREAL;
	r_offset_t3_dec_el:LREAL;
	l_offset_t1_acc_el:LREAL;
	l_offset_t2_v_el:LREAL;
	l_offset_t3_dec_el:LREAL;
	r_offset_t:LREAL:=0;
	test_t:LREAL;
	r_az_offset_abs:LREAL;
	
	Static_done: BOOL;
	r_write_position_az_s: LREAL;
	r_write_position_el_s: LREAL;
	s_mp: StaticPmParam;
	Az_rad: LREAL;
	El_rad: LREAL;
	ABphi_rad: LREAL;
	TE: INT;
	//r_write_position_az_out: LREAL;
	//r_write_position_el_out: LREAL;
	test1: BOOL;
	Test2: BOOL;
	test3: BOOL;
	test4: BOOL;
	test5: BOOL;
	test6: BOOL;
	test7: BOOL;
	test8: BOOL;
	test9: BOOL;
	rtrig_write_position_sim: R_TRIG;
	fb_move_sim_track_Az: MC_MoveAbsolute;
	b_sim_trk_az_done: BOOL;
	b_sim_trk_el_done: BOOL;
	rtrig_reset_sim: R_TRIG;
	rtrig_reset_sim_move: R_TRIG;
	fb_move_sim_track_El: MC_MoveAbsolute;
	b_sim_write_az: BOOL;
	b_sim_trk_az_active: BOOL;
	TON_0: TON;
	b_sim_trk_el_active: BOOL;
	b_sim_trk_az_active_not: BOOL;
	f_trig_sim: F_TRIG;
	R_TRIG_0: R_TRIG;
	F_TRIG_0: F_TRIG;
	F_TRIG_1: F_TRIG;
	TON_1: TON;
	IL_EnableInOpBase_0: IL_SIGNALGENERATORTYPE01;
	TP_0: TP;
	TP_1: TP;
	TP_2: TP;
	BLINK_0: BLINK;
	b_sim_trk_exec: BOOL;
END_VAR

(*IF test_enable_el THEN
arAxisCtrl_gb[Drive3.AxisNo].Admin._OpMode.en := Modeah;
ELSE
arAxisCtrl_gb[Drive3.AxisNo].Admin._OpMode.en := Modeab;
END_IF
*)
//axisdata[3].dwUserCmdDataA_q.REAL_;

//axisdata[3].dwUserActualDataA_i.REAL_;



//axisdata[3].dwUserCmdDataA_q.REAL_:=axisdata[3].dwUserActualDataA_i.REAL_;





(*<<<<<<<<<<<<<<<<<<<<<calculate the current point in the stack>>>>>>>>>>>>>>>>>>>>>>>*)
//WHILE lr_MJD_current >= track_table[F_I_number(i_start+1)].MJD DO
test1:=lr_TAIoffset_current >= track_table[F_I_number(i_start+1)].TAIoffset;
WHILE lr_TAIoffset_current >= track_table[F_I_number(i_start+1)].TAIoffset DO
	IF i_start= i_end THEN
		EXIT;
	ELSE
		i_start:=F_I_number(i_start+1);
	END_IF;
END_WHILE


(*<<<<<<<<<<<<<<<<<<calculate the number of the points left in the stack>>>>>>>>>>>>>>*)
IF i_start=i_end THEN
	i_num_stack_left:=0;
ELSE
	i_num_stack_left:= i_end-i_start+1;
	IF i_num_stack_left<=0 THEN
		i_num_stack_left:=i_num_stack_left+i_total;
	END_IF;
END_IF

(* I Don't know what this piece of code is meant to do commenting it out 8/8/2024
IF i_num_stack_left>10 AND b_remote_on_run AND b_track_on=FALSE THEN
	b_track_on:=TRUE;
END_IF; *)


r_abs_az_speed:=ABS(AxisData[1].rActualVelocity_i)*6;
p_covert_velocity:=(0.5773*r_abs_az_speed*r_abs_az_speed*r_abs_az_speed - 0.4526*r_abs_az_speed*r_abs_az_speed + 11.313*r_abs_az_speed + 4.523)*0.2535;
p_covert_velocity_el:=0.5773*r_vel_EL*r_vel_EL*r_vel_EL - 0.4526*r_vel_EL*r_vel_EL + 11.313*r_vel_EL + 4.523;
(*<<<<<<<<<<<<<<<<<<<<<<<<<<<<<<<<<<<<<<the definication of trigger and TON>>>>>>>>>>>>>>>>>>>>>>>>>>>>>>>>>>>>>>>>>>>>>>>*)
r_rtrig_start_stop(clk:=b_track_on);(*before tracking ,stop the motion*)
ton_track_on(IN:=b_track_on,PT:=T#200MS);(*by using 200ms,program can search about 60 points*)
rtrig_track_on(clk:=ton_track_on.Q);(*the trigger for the initializtion*)


ton_pause_on(IN:=b_Track_Pause,PT:=T#4000MS);(*by using 200ms,program can search about 60 points*)
rtrig_pause_on(clk:=ton_pause_on.Q);(*the trigger for the initializtion*)

IF rtrig_pause_on.Q THEN
	b_track_on:=FALSE;
END_IF


(*<<<<<<<<<<<<<<<<<<<<<<<<<<<<main program of track>>>>>>>>>>>>>>>>>>>>>>>>>>>>>*)
IF b_track_on=TRUE THEN
	
(*<<<<<<<<<<<<<<<<<<<<<<<<<<< Calculate the tracking error>>>>>>>>>>>>>>>>>>>>>>>>>>>>>*)
	
	//IF ABS(track_table[i_start].MJD-lr_mjd_current)*86400<0.001 THEN
	Test2:=ABS(track_table[i_start].TAIoffset-lr_TAIoffset_current)<0.001;
	IF ABS(track_table[i_start].TAIoffset-lr_TAIoffset_current)<0.001 THEN
		r_following_1:=(r_pos_az_v-track_table[i_start].Azimuth);
		IF  ABS(r_following_1)<0.5  THEN
		   r_following_1:=(r_pos_az_v-track_table[i_start].Azimuth)/p_covert_velocity;
		END_IF
		   r_following_3:=(r_pos_el_v-track_table[i_start].Elevation);
		IF ABS(r_following_3)>0.0001 AND ABS(r_following_3)<=0.003 THEN
			r_following_3:=(r_pos_el_v-track_table[i_start].Elevation)/1.5;
		END_IF
		IF ABS(r_following_3)>0.003 AND ABS(r_following_3)<=0.006 THEN
			r_following_3:=(r_pos_el_v-track_table[i_start].Elevation)/2;
		END_IF
		IF ABS(r_following_3)>0.006 AND ABS(r_following_3)<=0.02 THEN
			r_following_3:=(r_pos_el_v-track_table[i_start].Elevation)/4;
		END_IF
		r_following_radius_asec := LREAL_TO_REAL((SQRT(EXPT(r_following_1,2)+EXPT(r_following_3,2)))*3600);  // Following erroring terms of a radius. 
		
  (*      r_following_3:=(r_pos_el_v-track_table[i_start].Elevation_ori);
		IF ABS(r_following_3)>0.0001 AND ABS(r_following_3)<=0.003 THEN
			r_following_3:=(r_pos_el_v-track_table[i_start].Elevation_ori)/1.5;
		END_IF
		IF ABS(r_following_3)>0.003 AND ABS(r_following_3)<=0.006 THEN
			r_following_3:=(r_pos_el_v-track_table[i_start].Elevation_ori)/2;
		END_IF
		IF ABS(r_following_3)>0.006 AND ABS(r_following_3)<=0.02 THEN
			r_following_3:=(r_pos_el_v-track_table[i_start].Elevation_ori)/4;
		END_IF
		r_following_radius_asec := (SQRT(EXPT(r_following_1,2)+EXPT(r_following_3,2)))*3600;  // Following erroring terms of a radius. 
		*)
	END_IF
(*
	IF ABS(r_following_3)> ABS(r_track_error[2]) THEN	
		r_following_33:=r_track_error[2];
	ELSE
		r_following_33:=r_following_33;
	END_IF
		IF ABS(r_following_33)>0.01 THEN
			r_following_33:=r_following_33/10;
		END_IF
	IF ABS(r_vel_EL)<0.0001 THEN
		r_following_3:=r_following_33;
	ELSE
		r_following_3:=r_following_33/p_covert_velocity_el;
	END_IF	
*)	
(*<<<<<<<<<<<<when finish all the points or the power is down,then reset the track_on>>>>>>>>>>>>>>>>>>>*)
	IF i_start=i_end OR b_remote_on_run=FALSE THEN
		 b_track_on:=FALSE;
	END_IF
(*<<<<<<<<<<<<<<<<<<<<<<<<<<<<stop the motion before tracking>>>>>>>>>>>>>>>>>>>*)
	IF r_rtrig_start_stop.Q THEN
		b_SCC_STOP:=TRUE;
	END_IF
	IF rtrig_track_on.Q=TRUE THEN
(*<<<<<<<<<<<<<<<<<<<<<<<<<<<<<<find the first point which can be caught up>>>>>>>>>>>>>>>>>>>>>>>>>>>*)
		//WHILE ABS(track_table[i_start].Azimuth-r_pos_az_v)/((track_table[i_start].MJD-lr_mjd_current)*86400-0.05)>2.9 OR (track_table[i_start].MJD-lr_mjd_current)*86400-0.05<0 DO
		test3:=ABS(track_table[i_start].Azimuth-r_pos_az_v)/((track_table[i_start].TAIoffset-lr_TAIoffset_current)-0.05)>2.9 OR (track_table[i_start].TAIoffset-lr_TAIoffset_current)-0.05<0;
		WHILE ABS(track_table[i_start].Azimuth-r_pos_az_v)/((track_table[i_start].TAIoffset-lr_TAIoffset_current)-0.05)>2.9 OR (track_table[i_start].TAIoffset-lr_TAIoffset_current)-0.05<0 DO
		//WHILE ABS(entry_buffer1[i_start].Azimuth-r_pos_az_v)/((entry_buffer1[i_start].MJD-lr_mjd_current)*86400-0.05)>2.9 DO
			IF i_start=i_end-3 THEN
				EXIT;
			ELSE
				i_start:=F_I_number(i_start+1);
			END_IF
		END_WHILE
		
		//WHILE ABS(track_table[i_start].Elevation-r_pos_el)/((track_table[i_start].MJD-lr_mjd_current)*86400-0.05)>0.8 OR (track_table[i_start].MJD-lr_mjd_current)*86400-0.05<0 DO
		test4:=ABS(track_table[i_start].Elevation-r_pos_el)/((track_table[i_start].TAIoffset-lr_TAIoffset_current)-0.05)>0.8 OR (track_table[i_start].TAIoffset-lr_TAIoffset_current)-0.05<0;
		WHILE ABS(track_table[i_start].Elevation-r_pos_el)/((track_table[i_start].TAIoffset-lr_TAIoffset_current)-0.05)>0.8 OR (track_table[i_start].TAIoffset-lr_TAIoffset_current)-0.05<0 DO	
		//WHILE ABS(entry_buffer1[i_start].Elevation-r_pos_motor3)/((entry_buffer1[i_start].MJD-lr_mjd_current)*86400-0.05)>1000 DO
			IF i_start=i_end-3 THEN
				EXIT;
			ELSE
				i_start:=F_I_number(i_start+1);
			END_IF
		END_WHILE
(*		WHILE ABS(entry_buffer1[i_start].FeedIndexer-r_pos_FI_v)/((entry_buffer1[i_start].MJD-lr_mjd_current)*86400-0.05)>2 OR (entry_buffer1[i_start].MJD-lr_mjd_current)*86400-0.05<0 DO
			IF i_start=i_end-3 THEN
				EXIT;
			ELSE
				i_start:=F_I_number(i_start+1);
			END_IF
		END_WHILE
*)

//		arAxisCtrl_gb[Drive3.AxisNo].Admin._OpMode.en := ModeCyclicVelocity; 
		b_write_el_vel:=TRUE;
		i_point_caught:=i_start;
		//i_caught_MJD1:=track_table[i_point_caught].MJD;
		 i_caught_TAIoffset1:=track_table[i_point_caught].TAIoffset;
		//i_caught_MJD2:=lr_MJD_current;
		i_caught_TAIoffset2:=lr_TAIoffset_current;
		r_start_az:=r_pos_az_v;
		r_caught_az:=track_table[i_point_caught].Azimuth;
		
(*if the first point which can be caught up is the last one£¬reset track_on*)
		IF i_start=i_end-3 THEN
			b_track_on:=FALSE;
		ELSE
			//track_table[F_I_number(i_start-1)].MJD:=lr_MJD_current+0.0000008;(*(69ms)after gunner change p41 from 0 to 100ms*)
			track_table[F_I_number(i_start-1)].TAIoffset:=lr_TAIoffset_current+0.0000008;(*(69ms)after gunner change p41 from 0 to 100ms*)
			track_table[F_I_number(i_start-1)].Azimuth:=r_pos_az_v;
			track_table[F_I_number(i_start-1)].elevation:=r_pos_el;
(*			entry_buffer1[F_I_number(i_start-1)].FeedIndexer:=r_pos_FI_v;  *)
		i_start:=F_I_number(i_start-1);
		r_write_position_az:=track_table[i_start].Azimuth;
		r_write_position_el:=track_table[i_start].Elevation;
(*		r_write_position_FI:=entry_buffer1[i_start].FeedIndexer;   *)
		r_last_position_az:=r_write_position_az;
		r_last_position_el:=r_write_position_el;
(*		r_last_position_FI:=r_write_position_FI;   *)
		b_signal_for_open:=TRUE;
		END_IF

	END_IF
(*when the position is all nearby the start point,open the channel for writing position to all axis*)
test5:=b_signal_for_open AND (ABS(r_pos_az_v-track_table[i_start].Azimuth)<0.001) AND (ABS(r_pos_el-track_table[i_start].Elevation)<0.001);
	IF b_signal_for_open AND (ABS(r_pos_az_v-track_table[i_start].Azimuth)<0.001) AND (ABS(r_pos_el-track_table[i_start].Elevation)<0.001) THEN
		b_open_channel_az:=TRUE;
//		b_start_cyclicvel:=TRUE;
//		b_open_channel_el:=TRUE;
(*		b_open_channel_FI:=TRUE;*)
		b_signal_for_open:=FALSE;
	END_IF
(*defind the variables for calculating the cubic fuction*)
		//t:=lr_MJD_current;
		//t1:=track_table[i_start].MJD;
		//t2:=track_table[F_I_number(i_start+1)].MJD;
		//t3:=track_table[F_I_number(i_start+2)].MJD;
		t:=lr_TAIoffset_current;
		t1:=track_table[i_start].TAIoffset;
		t2:=track_table[F_I_number(i_start+1)].TAIoffset;
		t3:=track_table[F_I_number(i_start+2)].TAIoffset;
		p1_az:=track_table[i_start].Azimuth;
		p2_az:=track_table[F_I_number(i_start+1)].Azimuth;
		p3_az:=track_table[F_I_number(i_start+2)].Azimuth;
		
		r_test1:=p1_az;
		r_test2:=p2_az;
		r_test3:=p3_az;
		
		p1_el:=track_table[i_start].elevation;
		p2_el:=track_table[F_I_number(i_start+1)].elevation;
		p3_el:=track_table[F_I_number(i_start+2)].elevation;		
(*		p1_FI:=entry_buffer1[i_start].FeedIndexer;
		p2_FI:=entry_buffer1[F_I_number(i_start+1)].FeedIndexer;
		p3_FI:=entry_buffer1[F_I_number(i_start+2)].FeedIndexer;
*)		
		//i_start;
		test_1:=F_I_number(i_start+1);
		test_2:=F_I_number(i_start+2);
(*construct the first cubic section by 2 points and 2 velocity*)
(*	IF	lr_MJD_current<entry_buffer1[i_point_caught].MJD AND lr_MJD_current>entry_buffer1[F_I_number(i_point_caught-1)].MJD THEN  *)
	//IF	lr_MJD_current<i_caught_MJD1 AND lr_MJD_current>i_caught_MJD2 THEN
test6:=lr_TAIoffset_current<i_caught_TAIoffset1 AND lr_TAIoffset_current>i_caught_TAIoffset2;
 IF	lr_TAIoffset_current<i_caught_TAIoffset1 AND lr_TAIoffset_current>i_caught_TAIoffset2 THEN	
	
		IF b_track_on THEN
			V_start_az:=(p3_az-p2_az)/(t3-t2);
			V_start_el:=(p3_el-p2_el)/(t3-t2);
(*			V_start_FI:=(p3_FI-p2_FI)/(t3-t2);  *)
			v0_az:=V_start_az;
			v0_el:=V_start_el;
(*			v0_FI:=V_start_FI;   *)
			b_test:=TRUE;
			b_start_to_compensate:=TRUE;

			a_az:=V_start_az/(t2-t1)/(t2-t1)-2*(p2_az-p1_az)/(t2-t1)/(t2-t1)/(t2-t1);
			b_az:=3*(p2_az-p1_az)/(t2-t1)/(t2-t1)-V_start_az/(t2-t1);
			a_el:=V_start_el/(t2-t1)/(t2-t1)-2*(p2_el-p1_el)/(t2-t1)/(t2-t1)/(t2-t1);
			b_el:=3*(p2_el-p1_el)/(t2-t1)/(t2-t1)-V_start_el/(t2-t1);
(*			a_FI:=V_start_FI/(t2-t1)/(t2-t1)-2*(p2_FI-p1_FI)/(t2-t1)/(t2-t1)/(t2-t1);
			b_FI:=3*(p2_FI-p1_FI)/(t2-t1)/(t2-t1)-V_start_FI/(t2-t1);
*)
			r_write_position_az:=a_az*(t-t1)*(t-t1)*(t-t1)+b_az*(t-t1)*(t-t1)+p1_az;
			r_write_position_el:=a_el*(t-t1)*(t-t1)*(t-t1)+b_el*(t-t1)*(t-t1)+p1_el;
(*			r_write_position_FI:=a_FI*(t-t1)*(t-t1)*(t-t1)+b_FI*(t-t1)*(t-t1)+p1_FI;   *)
		END_IF
	ELSE
		IF i_num_stack_left>2 THEN
			IF b_track_on THEN
(*<<<<<<<<<<<<<<<<<<<<<<<<<<<<<calculate the a and b in the function y=ax^3+bx^2+cx+d>>>>>>>>>>>>>>>>>>>>>>*)
(*y=a*(x-x1)^3+b*(x-x1)^2+c(x-x1)+d,   c=v0,  d=y1*)
			a_az:=((p3_az-p1_az)/(t3-t1)/(t3-t1)-(p2_az-p1_az)/(t2-t1)/(t2-t1)-v0_az/(t3-t1)+v0_az/(t2-t1))/(t3-t2);
			b_az:=((p3_az-p1_az)*(t2-t1)/(t3-t1)/(t3-t1)-(p2_az-p1_az)*(t3-t1)/(t2-t1)/(t2-t1)-v0_az*(t2-t1)/(t3-t1)+v0_az*(t3-t1)/(t2-t1))/(t2-t3);
			a_el:=((p3_el-p1_el)/(t3-t1)/(t3-t1)-(p2_el-p1_el)/(t2-t1)/(t2-t1)-v0_el/(t3-t1)+v0_el/(t2-t1))/(t3-t2);
			b_el:=((p3_el-p1_el)*(t2-t1)/(t3-t1)/(t3-t1)-(p2_el-p1_el)*(t3-t1)/(t2-t1)/(t2-t1)-v0_el*(t2-t1)/(t3-t1)+v0_el*(t3-t1)/(t2-t1))/(t2-t3);
(*			a_FI:=((p3_FI-p1_FI)/(t3-t1)/(t3-t1)-(p2_FI-p1_FI)/(t2-t1)/(t2-t1)-v0_FI/(t3-t1)+v0_FI/(t2-t1))/(t3-t2);
			b_FI:=((p3_FI-p1_FI)*(t2-t1)/(t3-t1)/(t3-t1)-(p2_FI-p1_FI)*(t3-t1)/(t2-t1)/(t2-t1)-v0_FI*(t2-t1)/(t3-t1)+v0_FI*(t3-t1)/(t2-t1))/(t2-t3);
*)
b_test:=FALSE;
			//IF lr_MJD_current>=track_table[i_start].MJD AND lr_MJD_current<=track_table[F_I_number(i_start+1)].MJD THEN
			test7:=lr_TAIoffset_current>=track_table[i_start].TAIoffset AND lr_TAIoffset_current<=track_table[F_I_number(i_start+1)].TAIoffset;
			IF lr_TAIoffset_current>=track_table[i_start].TAIoffset AND lr_TAIoffset_current<=track_table[F_I_number(i_start+1)].TAIoffset THEN
			
				r_write_position_az:=a_az*(t-t1)*(t-t1)*(t-t1)+b_az*(t-t1)*(t-t1)+v0_az*(t-t1)+p1_az;
				r_write_position_el:=a_el*(t-t1)*(t-t1)*(t-t1)+b_el*(t-t1)*(t-t1)+v0_el*(t-t1)+p1_el;
				r_cyclic_velocity_test:=(p2_el-p1_el)/(t2-t1)/86400;
				//r_cyclic_velocity_test:=(p2_el-p1_el)/(t2-t1);
				r_cyclic_velocity:=V0_el/86400;
				// r_cyclic_velocity:=V0_el;
(*				r_write_position_FI:=a_FI*(t-t1)*(t-t1)*(t-t1)+b_FI*(t-t1)*(t-t1)+v0_FI*(t-t1)+p1_FI;   *)
			END_IF
(*calculate the velocity of the last point*)
			//IF (lr_MJD_current-track_table[F_I_number(i_start+1)].MJD)*86400>=-0.002 AND (lr_MJD_current-track_table[F_I_number(i_start+1)].MJD)*86400<0 THEN
			test8:=(lr_TAIoffset_current-track_table[F_I_number(i_start+1)].TAIoffset)>=-0.002 AND (lr_TAIoffset_current-track_table[F_I_number(i_start+1)].TAIoffset)<0;
			IF (lr_TAIoffset_current-track_table[F_I_number(i_start+1)].TAIoffset)>=-0.002 AND (lr_TAIoffset_current-track_table[F_I_number(i_start+1)].TAIoffset)<0 THEN
				V0_az:=3*a_az*(t2-t1)*(t2-t1)+2*b_az*(t2-t1)+v0_az;
				V0_el:=3*a_el*(t2-t1)*(t2-t1)+2*b_el*(t2-t1)+v0_el;
(*				V0_FI:=3*a_FI*(t2-t1)*(t2-t1)+2*b_FI*(t2-t1)+v0_FI;    *)
			END_IF
			END_IF
		ELSE
(*<<<<<<<<<<<<<<<<<<<<<<<<run the last two points>>>>>>>>>>>>>>>>>>>>>>>>>>*)
			IF b_track_on THEN 
				//IF lr_MJD_current>=track_table[i_start].MJD AND lr_MJD_current<=track_table[F_I_number(i_start+1)].MJD THEN
				test9:= lr_TAIoffset_current>=track_table[i_start].TAIoffset AND lr_TAIoffset_current<=track_table[F_I_number(i_start+1)].TAIoffset;
				IF lr_TAIoffset_current>=track_table[i_start].TAIoffset AND lr_TAIoffset_current<=track_table[F_I_number(i_start+1)].TAIoffset THEN
				r_write_position_az:=(p2_az-p1_az)*(t-t1)/(t2-t1)+p1_az;
				r_write_position_el:=(p2_el-p1_el)*(t-t1)/(t2-t1)+p1_el;
(*				r_write_position_FI:=((p2_FI-p1_FI)*(t-t1)/(t2-t1)+p1_FI);     *)
				END_IF
			END_IF
		END_IF
	END_IF

	
IF b_start_to_compensate THEN
//	r_offset_el:=r_compensation_value_motor;
	r_write_position_az:=r_write_position_az+r_test_offset_az;
	r_write_position_el:=r_write_position_el+r_test_offset_el;
//	r_write_position_el:=r_write_position_el+r_offset_el;
END_IF
	
(*<<<<<<<<<<<<<<<<<<<<<<<<<limit the trajectory speed >>>>>>>>>>>>>>>>>>>>>>>>>*)
(*Because the program runs every 2ms,so wo can limit the position by the rule ¦¤y<v*¦¤t.*)
(*Azimuth trajectory speed limit is 5.1¡ã/s*)
		IF r_write_position_az-r_last_position_az>0.0031 THEN
				r_write_position_az:=r_last_position_az+0.0031;
				b_track_overspeed_az:=1;
			ELSIF r_write_position_az-r_last_position_az<-0.0031 THEN
				r_write_position_az:=r_last_position_az-0.0031;
				b_track_overspeed_az:=1;
			ELSE
				b_track_overspeed_az:=0;
			END_IF
(*Elevation trajectory speed limit is 1.05¡ã/s*)
			IF r_write_position_el-r_last_position_el>0.00091 THEN
				r_write_position_el:=r_last_position_el+0.00091;
				b_track_overspeed_el:=1;
			ELSIF r_write_position_el-r_last_position_el<-0.00091 THEN
				r_write_position_el:=r_last_position_el-0.00091;
				b_track_overspeed_el:=1;
			ELSE
				b_track_overspeed_el:=0;
			END_IF
(*
(*FeedIndexer trajectory speed limit is 2.1¡ã/s*)
			IF r_write_position_FI-r_last_position_FI>0.0042 THEN
				r_write_position_FI:=r_last_position_FI+0.0042;
				b_track_overspeed_FI:=1;
			ELSIF r_write_position_FI-r_last_position_FI<-0.0042 THEN
				r_write_position_FI:=r_last_position_FI-0.0042;
				b_track_overspeed_FI:=1;
			ELSE
				b_track_overspeed_FI:=0;
			END_IF
*)
			
			
(*register the velocity and position for calculate the speed limit and acceleration limit*)
			r_last_position_az:=r_write_position_az;
			r_last_position_el:=r_write_position_el;
(*			r_last_position_FI:=r_write_position_FI;   *)
(*<<<<<<<<<<<<<<<<<<<<<<<<close the cyclic channel and reset the track error>>>>>>>>>>>>>>>>>>>>>>>>>>*)
ELSE
(*close the cyclic channel*)
	b_open_channel_az:=FALSE;
	b_open_channel_el:=FALSE;
	b_start_to_compensate:=FALSE;
	r_compensation_value_motor:=0;
(*	b_open_channel_FI:=FALSE;  *)
(*reset the following error and so on*)
    r_write_position_el:= axisdata[8].rActualPosition_i;
	r_write_position_az:=  axisdata[7].rActualPosition_i;
	r_track_error[1]:=0;
	r_track_error[2]:=0;
	r_track_error[3]:=0;
	V0_az:=0;
	V0_el:=0;
	V_start_az:=0;
	V_start_el:=0;
	IF NOT(b_SCC_goto) AND NOT(b_track_on) THEN 
		r_following_1:=0.00;
		r_following_3:=0.00;
	END_IF
END_IF

 IF  b_test_offset_start THEN
	 	r_offset_t:=r_offset_t+0.001;
		test_t:=r_offset_t-r_offset_t1_acc-r_offset_t2_v;
 		(*****************AZ offset**********)
		r_az_offset_abs:=ABS(r_offset_az);
		r_offset_t1_acc:=r_az_offset_Vmax/r_az_offset_acc;
	 	r_offset_t3_dec:=r_az_offset_Vmax/r_az_offset_dec;
	 	l_offset_t1_acc:=0.5*r_az_offset_acc*r_offset_t1_acc*r_offset_t1_acc;
	 	l_offset_t3_dec:=0.5*r_az_offset_dec*r_offset_t3_dec*r_offset_t3_dec;
 		r_offset_t2_v:=(r_az_offset_abs-l_offset_t1_acc-l_offset_t3_dec)/r_az_offset_Vmax;
		l_offset_t2_v:=r_az_offset_Vmax*r_offset_t2_v;

			IF r_offset_t <=r_offset_t1_acc THEN
				r_test_offset_az_abs:=0.5*r_az_offset_acc*r_offset_t*r_offset_t;
			ELSIF r_offset_t1_acc<r_offset_t AND r_offset_t<(r_offset_t1_acc+r_offset_t2_v) THEN 
				r_test_offset_az_abs:=r_test_offset_az_abs+0.001*r_az_offset_Vmax;
			ELSIF (r_offset_t1_acc+r_offset_t2_v)<=r_offset_t AND r_offset_t<(r_offset_t1_acc+r_offset_t2_v+r_offset_t3_dec) THEN
				r_test_offset_az_abs:=l_offset_t1_acc+l_offset_t2_v+(r_offset_t-r_offset_t1_acc-r_offset_t2_v)*r_az_offset_Vmax-0.5*r_az_offset_dec*(r_offset_t-r_offset_t1_acc-r_offset_t2_v)*(r_offset_t-r_offset_t1_acc-r_offset_t2_v);
			ELSE 
				r_test_offset_az_abs:=r_az_offset_abs;
			END_IF

		IF r_test_offset_az_abs>=r_az_offset_abs THEN
			r_test_offset_az_abs:=r_az_offset_abs;
		END_IF
		IF r_offset_az<0 THEN
			r_test_offset_az:=-r_test_offset_az_abs;
		ELSE 
			r_test_offset_az:=r_test_offset_az_abs;
		END_IF
		r_test_offset_az:=r_offset_az_old+r_test_offset_az;
		
		
			(*****************EL offset**********)
		r_el_offset_abs:=ABS(r_offset_el);
		r_offset_t1_acc_el:=r_el_offset_Vmax/r_el_offset_acc;
	 	r_offset_t3_dec_el:=r_el_offset_Vmax/r_el_offset_dec;
	 	l_offset_t1_acc_el:=0.5*r_el_offset_acc*r_offset_t1_acc_el*r_offset_t1_acc_el;
	 	l_offset_t3_dec_el:=0.5*r_el_offset_dec*r_offset_t3_dec_el*r_offset_t3_dec_el;
 		r_offset_t2_v_el:=(r_el_offset_abs-l_offset_t1_acc_el-l_offset_t3_dec_el)/r_el_offset_Vmax;
		l_offset_t2_v_el:=r_el_offset_Vmax*r_offset_t2_v_el;

			IF r_offset_t <=r_offset_t1_acc_el THEN
				r_test_offset_el_abs:=0.5*r_el_offset_acc*r_offset_t*r_offset_t;
			ELSIF r_offset_t1_acc_el<r_offset_t AND r_offset_t<(r_offset_t1_acc_el+r_offset_t2_v_el) THEN 
				r_test_offset_el_abs:=r_test_offset_el_abs+0.001*r_el_offset_Vmax;
			ELSIF (r_offset_t1_acc_el+r_offset_t2_v_el)<=r_offset_t AND r_offset_t<(r_offset_t1_acc_el+r_offset_t2_v_el+r_offset_t3_dec_el) THEN
				r_test_offset_el_abs:=l_offset_t1_acc_el+l_offset_t2_v_el+(r_offset_t-r_offset_t1_acc_el-r_offset_t2_v_el)*r_el_offset_Vmax-0.5*r_el_offset_dec*(r_offset_t-r_offset_t1_acc_el-r_offset_t2_v_el)*(r_offset_t-r_offset_t1_acc_el-r_offset_t2_v_el);
			ELSE 
				r_test_offset_el_abs:=r_el_offset_abs;
			END_IF

		IF r_test_offset_el_abs>=r_el_offset_abs THEN
			r_test_offset_el_abs:=r_el_offset_abs;
		END_IF
		IF r_offset_el<0 THEN
			r_test_offset_el:=-r_test_offset_el_abs;
		ELSE 
			r_test_offset_el:=r_test_offset_el_abs;
		END_IF
		r_test_offset_el:=r_offset_el_old+r_test_offset_el;
    IF 	r_test_offset_el_abs=r_el_offset_abs AND r_test_offset_az_abs=r_az_offset_abs THEN 	
		b_test_offset_start:=FALSE;
		b_offset_running:=FALSE;
	END_IF
				
ELSE
	i_test_offset_count:=0;
	r_offset_t:=0;
	r_offset_az_old:=r_test_offset_az;
	r_offset_el_old:=r_test_offset_el;
END_IF


P_Track_cubic.A_StaticPM();
P_Track_cubic.A_AmbTempPM();
P_Track_cubic.A_DynamicPM();


Tracking.Status.p_desired_El:=r_write_position_el-Tracking.Status.act_statOffset_value_El/gc_lr_arcsec2deg;
Tracking.Status.p_desired_Az:=r_write_position_az-(Tracking.Status.act_statOffset_value_Xel/gc_lr_arcsec2deg)/COS(ML_degtorad(r_write_position_el));

IF b_track_on THEN 
r_write_position_az_out:=r_write_position_az-Pointing.Status.StaticPmCorrVal_Az/gc_lr_arcsec2deg-Pointing.Status.TiltCorrVal_Az/gc_lr_arcsec2deg-Pointing.Status.AmbTempCorrVal_Az/gc_lr_arcsec2deg;
r_write_position_el_out:=r_write_position_el-Pointing.Status.StaticPmCorrVal_El/gc_lr_arcsec2deg-Pointing.Status.TiltCorrVal_El/gc_lr_arcsec2deg-Pointing.Status.AmbTempCorrVal_El/gc_lr_arcsec2deg;
END_IF

IF gc_b_sim_on THEN 
	P_Track_cubic.A_Sim_track_function_blocks();
ELSE	
	P_Track_cubic.A_track_fuction_blocks();
END_IF

ACTION A_track_fuction_blocks:
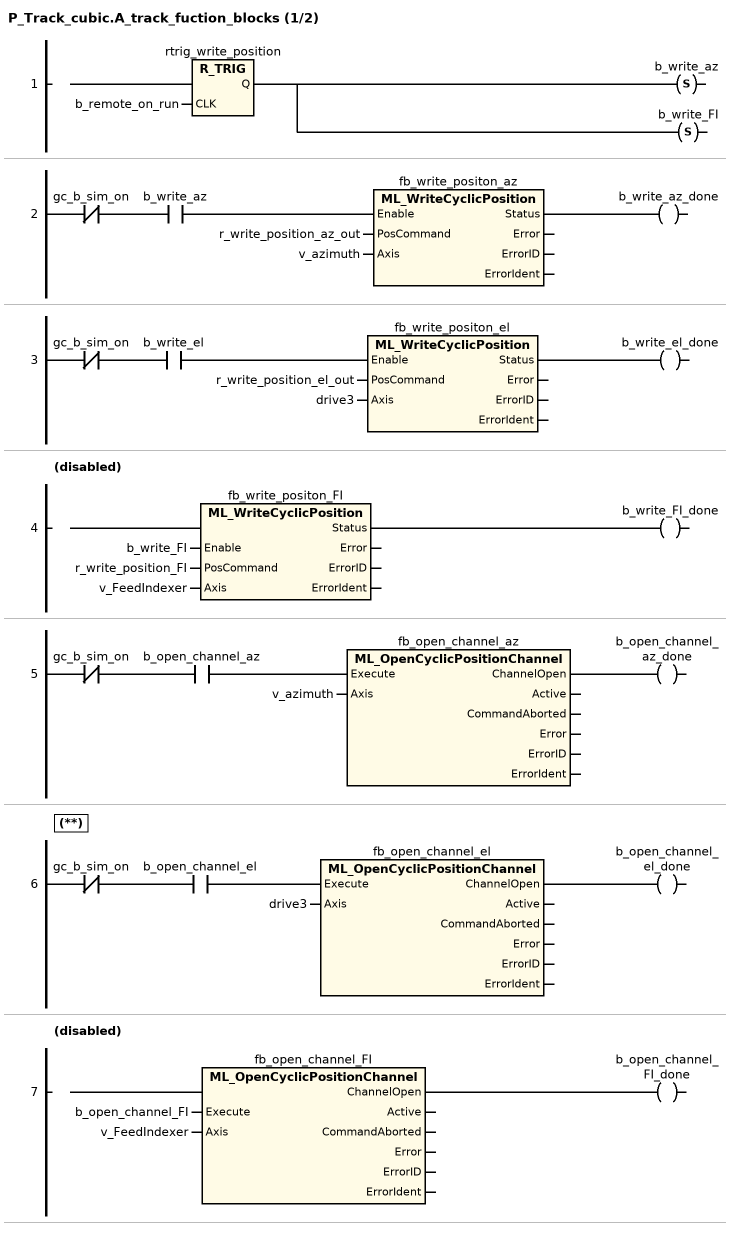
// NETWORK 1
rtrig_write_position(CLK := b_remote_on_run); // R_TRIG
b_write_az S= rtrig_write_position.Q;
b_write_FI S= rtrig_write_position.Q;

// NETWORK 2
fb_write_positon_az(
    Enable := NOT gc_b_sim_on AND b_write_az,
    PosCommand := r_write_position_az_out,
    Axis := v_azimuth); // ML_WriteCyclicPosition
b_write_az_done := fb_write_positon_az.Status;

// NETWORK 3
fb_write_positon_el(
    Enable := NOT gc_b_sim_on AND b_write_el,
    PosCommand := r_write_position_el_out,
    Axis := drive3); // ML_WriteCyclicPosition
b_write_el_done := fb_write_positon_el.Status;

// NETWORK 4 (disabled)
// fb_write_positon_FI(Enable := b_write_FI, PosCommand := r_write_position_FI, Axis := v_FeedIndexer); // ML_WriteCyclicPosition
// b_write_FI_done := fb_write_positon_FI.Status;

// NETWORK 5
fb_open_channel_az(Execute := NOT gc_b_sim_on AND b_open_channel_az, Axis := v_azimuth); // ML_OpenCyclicPositionChannel
b_open_channel_az_done := fb_open_channel_az.ChannelOpen;

// NETWORK 6
// label: (**)
fb_open_channel_el(Execute := NOT gc_b_sim_on AND b_open_channel_el, Axis := drive3); // ML_OpenCyclicPositionChannel
b_open_channel_el_done := fb_open_channel_el.ChannelOpen;

// NETWORK 7 (disabled)
// fb_open_channel_FI(Execute := b_open_channel_FI, Axis := v_FeedIndexer); // ML_OpenCyclicPositionChannel
// b_open_channel_FI_done := fb_open_channel_FI.ChannelOpen;

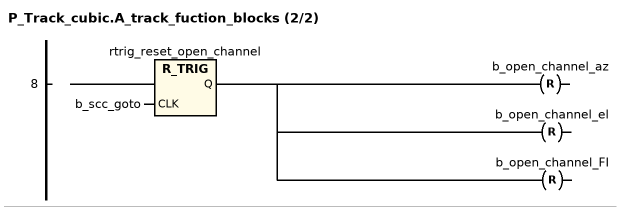
// NETWORK 8
rtrig_reset_open_channel(CLK := b_scc_goto); // R_TRIG
b_open_channel_az R= rtrig_reset_open_channel.Q;
b_open_channel_el R= rtrig_reset_open_channel.Q;
b_open_channel_FI R= rtrig_reset_open_channel.Q;
END_ACTION

ACTION A_StaticPM:
s_mp:= Pointing.StaticPmParameters[Pointing.Status.BandForCorr]; 

// Convert to Radians for trigonometric functions. 
Az_rad:= ML_degtorad(r_write_position_az);
IF r_write_position_el>= 85 THEN
	El_rad:= ML_degtorad(85);
ELSE
	El_rad:= ML_degtorad(r_write_position_el);	
END_IF

ABphi_rad:=ML_degtorad(s_mp.ABphi);

IF Pointing.Status.StaticCorrActive = 1 THEN 
	IF pointing.Status.TiltCorrActive = 1 THEN 
	// Calc Pointing correction with gravity tilt removed
	   TE := 0;
	ELSE 
	// Calc Pointing correction with gravity tilt
	   TE :=1;
    END_IF
	
	 Pointing.Status.StaticPmCorrVal_Az := ( -s_mp.IA - s_mp.CA/COS(El_rad) - s_mp.NPAE*TAN(El_rad) - s_mp.AN*SIN(Az_rad)*TAN(El_rad) - s_mp.AW*COS(Az_rad)*TAN(El_rad) + s_mp.ACEC*COS(Az_rad)
      - s_mp.ACES*SIN(Az_rad) - s_mp.ABA*SIN(ABphi_rad)*COS(2*Az_rad)*(1-TE) +   s_mp.ABA*COS(ABphi_rad)*SIN(2*Az_rad)*(1-TE) + Tracking.Status.act_statOffset_value_Xel/COS(El_rad) +
     (s_mp.AN0*SIN(Az_rad)*TAN(El_rad) + s_mp.AW0*COS(Az_rad)*TAN(El_rad))*TE);
	 
	(* Tiltmeter correction included in static pointing model.
       Pointing.Status.StaticPmCorrVal_Az :=  -s_mp.IA - s_mp.CA/COS(El) - s_mp.NPAE*TAN(El) - s_mp.AN*SIN(Az)*TAN(El) - s_mp.AW*COS(Az)*TAN(El) + s_mp.ACEC*COS(Az)
      - s_mp.ACES*SIN(Az) - s_mp.ABA*SIN(s_mp.ABphi)*COS(2*Az)*(1-TE) +   s_mp.ABA*COS(s_mp.ABphi)*SIN(2*Az)*(1-TE) + Tracking.Status.act_statOffset_value_Xel/COS(El) +
     (ΔAz_tiltmeter + s_mp.AN0*SIN(Az)*TAN(El) + s_mp.AW0*COS(Az)*TAN(El))*TE; *)
	
	Pointing.Status.StaticPmCorrVal_El := (s_mp.IE - s_mp.AN*COS(Az_rad) +s_mp.AW*SIN(Az_rad)+ s_mp.ECEC*COS(El_rad) + s_mp.ECES*SIN(El_rad) + s_mp.ABA*COS(ABphi_rad)*COS(2*Az_rad)*(1-TE) + s_mp.ABA*SIN(ABphi_rad)*SIN(2*Az_rad)*(1-TE) + 
    s_mp.HECE4*COS(4*El_rad) + s_mp.HESE4*SIN(4*El_rad) + s_mp.HECE8*COS(8*El_rad) + s_mp.HESE8*SIN(8*El_rad) + Tracking.Status.act_statOffset_value_El +
    (s_mp.AN0*COS(Az_rad) - s_mp.AW0*SIN(Az_rad))*TE);
	(*  Tiltmeter correction included in static pointing model.
	 Pointing.Status.StaticPmCorrVal_El := s_mp.IE - s_mp.AN*COS(Az) +s_mp.AW*SIN(Az)+ s_mp.ECEC*COS(El) + s_mp.ECES*SIN(El) + s_mp.ABA*COS(s_mp.ABphi)*COS(2*Az)*(1-TE) + s_mp.ABA*SIN(ABphi)*SIN(2*Az)*(1-TE) + 
    s_mp.HECE4*COS(4*El) + s_mp.HESE4*SIN(4*El) + s_mp.HECE8*COS(8*El) + s_mp.HESE8*SIN(8*El) + Tracking.Status.act_statOffset_value_El +
    (ΔEl_tiltmeter + s_mp.AN0*COS(Az) - s_mp.AW0*SIN(Az))*TE; *)
   
ELSE 
// No calculation of static model only offsets
   Pointing.Status.StaticPmCorrVal_Az := (Tracking.Status.act_statOffset_value_Xel/COS(El_rad));
   Pointing.Status.StaticPmCorrVal_El := Tracking.Status.act_statOffset_value_El;
END_IF


IF   ABS(Pointing.Status.StaticPmCorrVal_Az) > gc_lr_point_corr_error_lim OR  ABS(Pointing.Status.StaticPmCorrVal_El) > gc_lr_point_corr_error_lim THEN 
   Pointing.Status.StaticPmCorrVal_Az := 0; 
   Pointing.Status.StaticPmCorrVal_El := 0;
   Management.ErrorStatus.errPoint := 1; 
END_IF
END_ACTION

ACTION A_DynamicPM:
	IF Pointing.Status.TiltOne_On THEN 
    	Pointing.Status.TiltCorrVal_Az:= Pointing.Status.TiltYArcsec_One*TAN(El_rad); //El_rad is calculated in the Stati PM section 
		Pointing.Status.TiltCorrVal_El:= Pointing.Status.TiltXArcsec_One;
	ELSIF Pointing.Status.TiltTwo_On THEN
		Pointing.Status.TiltCorrVal_Az:= Pointing.Status.TiltYArcsec_One*TAN(El_rad);
		Pointing.Status.TiltCorrVal_El:= Pointing.Status.TiltXArcsec_One;
	ELSE
		Pointing.Status.TiltCorrVal_Az:= 0;
		Pointing.Status.TiltCorrVal_El:= 0;
	END_IF

//	Check velocity
IF  ABS(axisdata[1].rActualVelocity_i)>= gc_r_tilt_vel_limit_Az THEN 
	Pointing.Status.TiltCorrVal_Az:= 0;
    Pointing.Status.TiltCorrVal_El:= 0;
END_IF

// Check if the correction is with in limits 
// The behaviour if the correction is outside the limits still needs to be finalised
IF ABS(Pointing.Status.TiltCorrVal_Az)>= gc_lr_tilt_corr_limit_Az OR ABS(Pointing.Status.TiltCorrVal_El)>=gc_lr_tilt_corr_limit_El THEN 
	Pointing.Status.TiltCorrVal_Az:= gc_lr_tilt_corr_limit_Az;
    Pointing.Status.TiltCorrVal_El:= gc_lr_tilt_corr_limit_El;
END_IF
END_ACTION

ACTION A_AmbTempPM:
IF Pointing.Status.AmbTempCorrActive THEN 
	Pointing.Status.AmbTempCorrVal_Az:=0;
	Pointing.Status.AmbTempCorrVal_El:=0;
ELSE
	Pointing.Status.AmbTempCorrVal_Az:=0;
	Pointing.Status.AmbTempCorrVal_El:=0;
END_IF
END_ACTION

ACTION A_Sim_track_function_blocks:
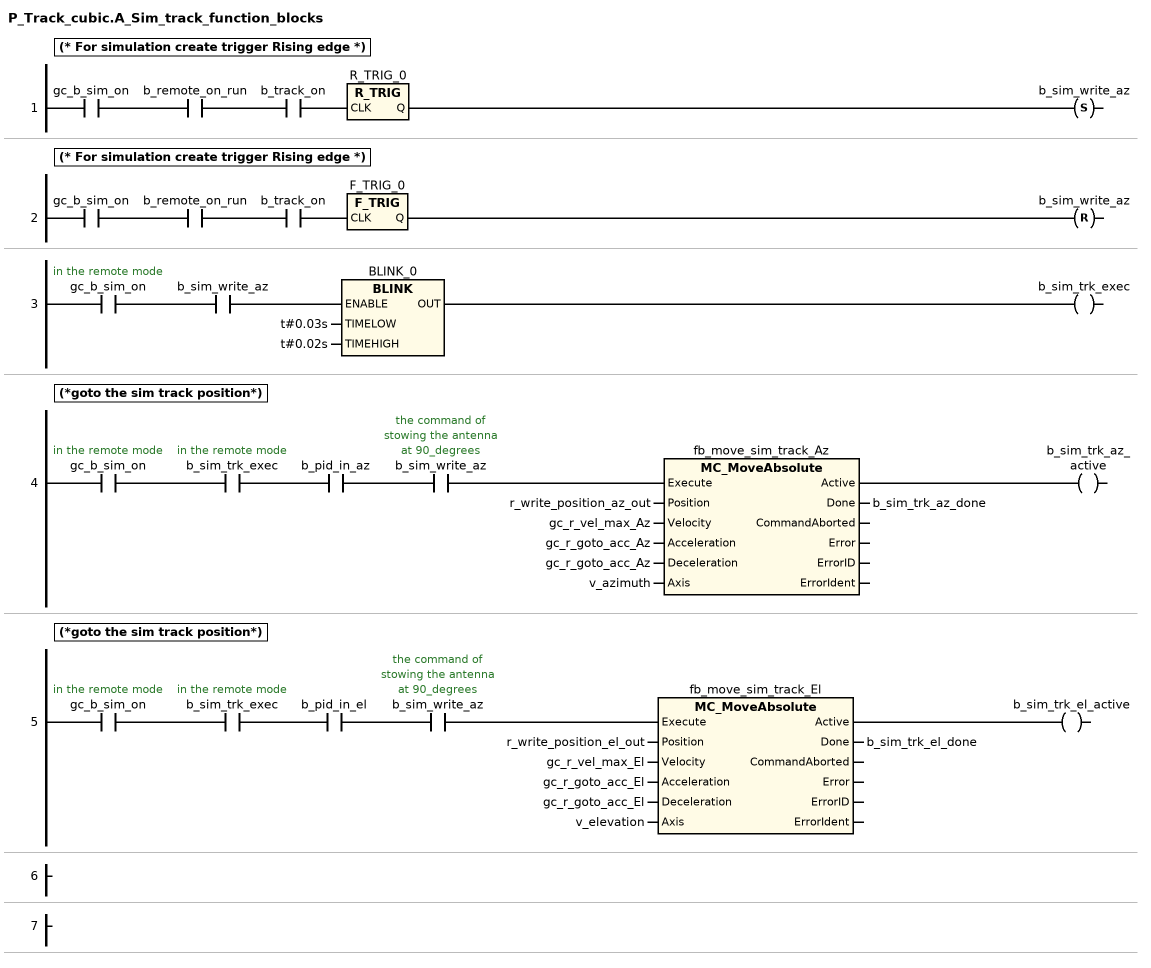
// NETWORK 1
// label: (* For simulation create trigger Rising edge *)
R_TRIG_0(CLK := gc_b_sim_on AND b_remote_on_run AND b_track_on); // R_TRIG
b_sim_write_az S= R_TRIG_0.Q;

// NETWORK 2
// label: (* For simulation create trigger Rising edge *)
F_TRIG_0(CLK := gc_b_sim_on AND b_remote_on_run AND b_track_on); // F_TRIG
b_sim_write_az R= F_TRIG_0.Q;

// NETWORK 3
//   gc_b_sim_on: in the remote mode
BLINK_0(ENABLE := gc_b_sim_on AND b_sim_write_az, TIMELOW := t#0.03s, TIMEHIGH := t#0.02s); // BLINK
b_sim_trk_exec := BLINK_0.OUT;

// NETWORK 4
//   fb_move_sim_track_Az: move the elevation to the fixed position
//   gc_b_sim_on: in the remote mode
//   b_sim_trk_exec: in the remote mode
//   b_sim_write_az: the command of stowing the antenna at 90_degrees
//   v_azimuth: Virtual axis "v_elevation" with axis number 8
// label: (*goto the sim track position*)
fb_move_sim_track_Az(
    Execute := gc_b_sim_on AND b_sim_trk_exec AND b_pid_in_az AND b_sim_write_az,
    Position := r_write_position_az_out,
    Velocity := gc_r_vel_max_Az,
    Acceleration := gc_r_goto_acc_Az,
    Deceleration := gc_r_goto_acc_Az,
    Axis := v_azimuth,
    Done => b_sim_trk_az_done); // MC_MoveAbsolute
b_sim_trk_az_active := fb_move_sim_track_Az.Active;

// NETWORK 5
//   fb_move_sim_track_El: move the elevation to the fixed position
//   gc_b_sim_on: in the remote mode
//   b_sim_trk_exec: in the remote mode
//   b_sim_write_az: the command of stowing the antenna at 90_degrees
//   v_elevation: Virtual axis "v_elevation" with axis number 8
// label: (*goto the sim track position*)
fb_move_sim_track_El(
    Execute := gc_b_sim_on AND b_sim_trk_exec AND b_pid_in_el AND b_sim_write_az,
    Position := r_write_position_el_out,
    Velocity := gc_r_vel_max_El,
    Acceleration := gc_r_goto_acc_El,
    Deceleration := gc_r_goto_acc_El,
    Axis := v_elevation,
    Done => b_sim_trk_el_done); // MC_MoveAbsolute
b_sim_trk_el_active := fb_move_sim_track_El.Active;

// NETWORK 6

// NETWORK 7
END_ACTION

END_PROGRAM

// IndraMotionMlc1/Application/POUs/TCP/Message/F_I_number
(*This program is bulit for transforming a minus value to a plus value*)
FUNCTION F_I_number : UINT
VAR_INPUT
	I_number:INT;
END_VAR
VAR
END_VAR

IF i_number <= 0 THEN
	i_number:=i_number+i_total;
END_IF;

IF i_number>i_total THEN
	i_number:=i_number-i_total;
END_IF;
F_I_number:=i_number;

END_FUNCTION

// IndraMotionMlc1/Application/POUs/Motion/P_power_on_TCP
(*the program is built for power on the 3 axis under the contol of remote or local.
the elevation axis is the similar with the azimuth*)
PROGRAM P_power_on_TCP
VAR
(*<<<<<<<<definition of r_trig for detecting a rising edge>>>>>>>>>>>>>>*)
	fb_rtrig_p1: R_TRIG;
	fb_rtrig_p3: R_TRIG;
	fb_rtrig_p5: R_TRIG;
	fb_rtrig_az: R_TRIG;
	fb_rtrig_el: R_TRIG;
	fb_rtrig_FI: R_TRIG;
	fb_rtrig_en_remote: R_TRIG;
	fb_rtrig_en_TCP: R_TRIG;
(*<<<<<<<The function block Timer On Delay implements a turn-on delay>>>>>>*)
	ton_en_1: TON;
	ton_en_2: TON;
	ton_en_3: TON;
	ton_en_4: TON;
	ton_en_5: TON;
	ton_en_6: TON;
(*MC_Power function block controls the power connection (power on or off)*)
	FB_1_power: MC_Power;
	FB_2_power: MC_Power;
	FB_3_power: MC_Power;
	FB_4_power: MC_Power;
	FB_5_power: MC_Power;
	FB_6_power: MC_Power;
	b_1_enable_on: BOOL;
	b_2_enable_on: BOOL;
	b_3_enable_on: BOOL;
	b_4_enable_on: BOOL;
	b_5_enable_on: BOOL;
	b_6_enable_on: BOOL;
(*With "MB_GearInPos",it is possible to realize a motion of the slave axis which is phase synchronous to the master axis*)
	fb_gearinPos_1: MB_GearInPos;
	fb_gearin_2: MB_GearInPos;
	fb_gearinPos_3: MB_GearInPos;
	fb_gearin_4: MB_GearInPos;
	fb_gearinPos_5: MB_GearInPos;
	fb_gearin_6: MB_GearInPos;
	b_gearin_1_done: BOOL;
	
	b_gearin_5_done:BOOL;
(*"MC_MoveAbsolute" is used to move the drive to a preset absolute position.*)
	FB_move_master_az: MC_MoveAbsolute;
	FB_move_master_el: MC_MoveAbsolute;
	FB_move_master_FI: MC_MoveAbsolute;
	b_M_az_done: BOOL;
	b_M_el_done: BOOL;
	b_M_FI_done: BOOL;
(*MB_Home function block controls axes with incremental encoder when executing the "search home" sequence*)
	fb_home_az2: MB_Home;
	fb_home_el2: MB_Home;
	fb_home_FI2: MB_Home;
	b_home_az2_done: BOOL;
	b_home_el2_done: BOOL;
	b_home_FI2_done: BOOL;
(*<<<<<<<<<<<<<<<<<<<<<<<<<<<<<clear error>>>>>>>>>>>>>>>>>>>>>>>>>>>>>>>>>*)
	TCP_clear_error: BOOL;
	FB_clear_error_TCP: MB_WriteParameter;
	TCP_clear_done: BOOL;
(*add 2011 06 09 to delete 1sec delay*)
	fb_gearinPos_el: MB_GearInPos;
	b_gearin_el_done: BOOL;
	fb_gearout_el: MC_GearOut;
	rtrig_set_gearin_3: R_TRIG;
	b_gearin_3: BOOL;
	rtrig_reset_gearin_3: F_TRIG;
	ton_clear_on: TON;
	fb_gearinPos_FI: MB_GearInPos;
	test_111: BOOL;
	ssss: BOOL;
	test1: BOOL;
	test2: BOOL;
	test3: BOOL;
	TON_enable_az: ton;
	TON_enable_az2: ton;
END_VAR

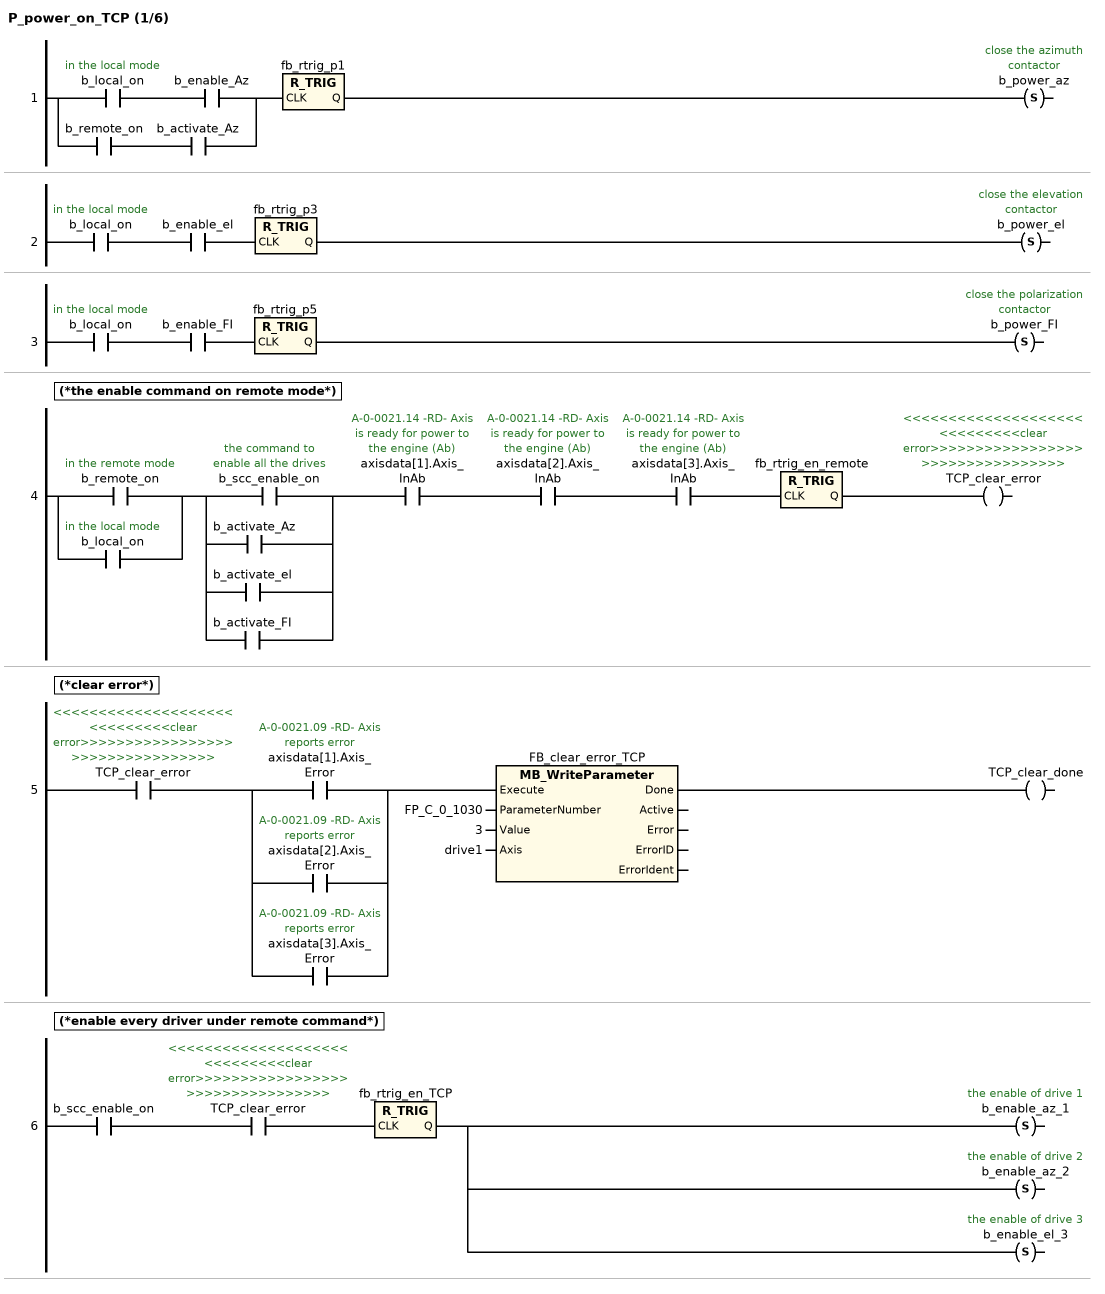
// NETWORK 1
//   fb_rtrig_p1: <<<<<<<<definition of r_trig for detecting a rising edge>>>>>>>>>>>>>>
//   b_local_on: in the local mode
//   b_power_az: close the azimuth contactor
fb_rtrig_p1(CLK := b_local_on AND b_enable_Az OR b_remote_on AND b_activate_Az); // R_TRIG
b_power_az S= fb_rtrig_p1.Q;

// NETWORK 2
//   b_local_on: in the local mode
//   b_power_el: close the elevation contactor
fb_rtrig_p3(CLK := b_local_on AND b_enable_el); // R_TRIG
b_power_el S= fb_rtrig_p3.Q;

// NETWORK 3
//   b_local_on: in the local mode
//   b_power_FI: close the polarization contactor
fb_rtrig_p5(CLK := b_local_on AND b_enable_FI); // R_TRIG
b_power_FI S= fb_rtrig_p5.Q;

// NETWORK 4
//   b_remote_on: in the remote mode
//   b_local_on: in the local mode
//   b_scc_enable_on: the command to enable all the drives
//   axisdata[1].Axis_InAb: A-0-0021.14 -RD- Axis is ready for power to the engine (Ab)
//   axisdata[2].Axis_InAb: A-0-0021.14 -RD- Axis is ready for power to the engine (Ab)
//   axisdata[3].Axis_InAb: A-0-0021.14 -RD- Axis is ready for power to the engine (Ab)
//   TCP_clear_error: <<<<<<<<<<<<<<<<<<<<<<<<<<<<<clear error>>>>>>>>>>>>>>>>>>>>>>>>>>>>>>>>>
// label: (*the enable command on remote mode*)
fb_rtrig_en_remote(CLK := (b_remote_on OR b_local_on) AND (b_scc_enable_on OR b_activate_Az OR b_activate_el OR b_activate_FI) AND axisdata[1].Axis_InAb AND axisdata[2].Axis_InAb AND axisdata[3].Axis_InAb); // R_TRIG
TCP_clear_error := fb_rtrig_en_remote.Q;

// NETWORK 5
//   TCP_clear_error: <<<<<<<<<<<<<<<<<<<<<<<<<<<<<clear error>>>>>>>>>>>>>>>>>>>>>>>>>>>>>>>>>
//   axisdata[1].Axis_Error: A-0-0021.09 -RD- Axis reports error
//   axisdata[2].Axis_Error: A-0-0021.09 -RD- Axis reports error
//   axisdata[3].Axis_Error: A-0-0021.09 -RD- Axis reports error
//   FP_C_0_1030: Command: Clear all control errors
//   drive1: Real axis "Drive1" with axis number 1
// label: (*clear error*)
FB_clear_error_TCP(
    Execute := TCP_clear_error AND (axisdata[1].Axis_Error OR axisdata[2].Axis_Error OR axisdata[3].Axis_Error),
    ParameterNumber := FP_C_0_1030,
    Value := 3,
    Axis := drive1); // MB_WriteParameter
TCP_clear_done := FB_clear_error_TCP.Done;

// NETWORK 6
//   TCP_clear_error: <<<<<<<<<<<<<<<<<<<<<<<<<<<<<clear error>>>>>>>>>>>>>>>>>>>>>>>>>>>>>>>>>
//   b_enable_az_1: the enable of drive 1
//   b_enable_az_2: the enable of drive 2
//   b_enable_el_3: the enable of drive 3
// label: (*enable every driver under remote command*)
fb_rtrig_en_TCP(CLK := b_scc_enable_on AND TCP_clear_error); // R_TRIG
b_enable_az_1 S= fb_rtrig_en_TCP.Q;
b_enable_az_2 S= fb_rtrig_en_TCP.Q;
b_enable_el_3 S= fb_rtrig_en_TCP.Q;

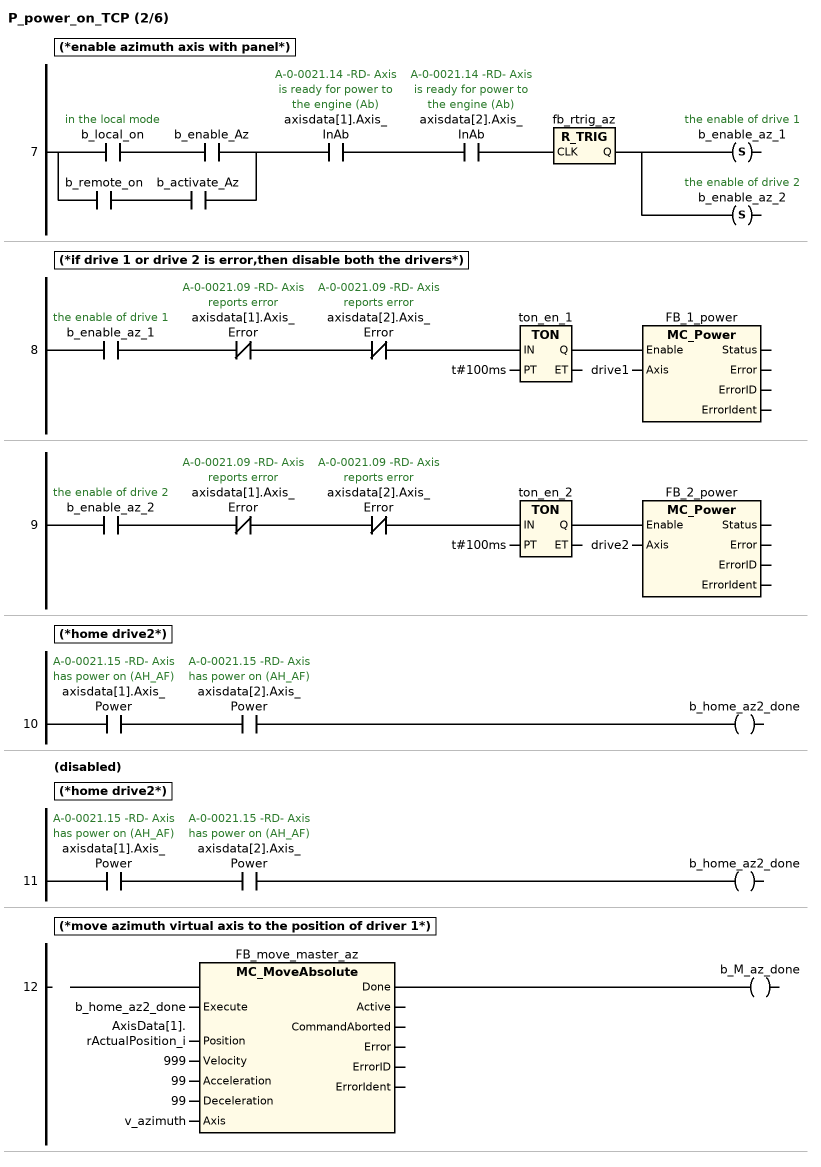
// NETWORK 7
//   b_local_on: in the local mode
//   axisdata[1].Axis_InAb: A-0-0021.14 -RD- Axis is ready for power to the engine (Ab)
//   axisdata[2].Axis_InAb: A-0-0021.14 -RD- Axis is ready for power to the engine (Ab)
//   b_enable_az_1: the enable of drive 1
//   b_enable_az_2: the enable of drive 2
// label: (*enable azimuth axis with panel*)
fb_rtrig_az(CLK := (b_local_on AND b_enable_Az OR b_remote_on AND b_activate_Az) AND axisdata[1].Axis_InAb AND axisdata[2].Axis_InAb); // R_TRIG
b_enable_az_1 S= fb_rtrig_az.Q;
b_enable_az_2 S= fb_rtrig_az.Q;

// NETWORK 8
//   FB_1_power: MC_Power function block controls the power connection (power on or off)
//   ton_en_1: <<<<<<<The function block Timer On Delay implements a turn-on delay>>>>>>
//   b_enable_az_1: the enable of drive 1
//   axisdata[1].Axis_Error: A-0-0021.09 -RD- Axis reports error
//   axisdata[2].Axis_Error: A-0-0021.09 -RD- Axis reports error
//   drive1: Real axis "Drive1" with axis number 1
// label: (*if drive 1 or drive 2 is error,then disable both the drivers*)
ton_en_1(IN := b_enable_az_1 AND NOT axisdata[1].Axis_Error AND NOT axisdata[2].Axis_Error, PT := t#100ms); // TON
FB_1_power(Enable := ton_en_1.Q, Axis := drive1); // MC_Power

// NETWORK 9
//   b_enable_az_2: the enable of drive 2
//   axisdata[1].Axis_Error: A-0-0021.09 -RD- Axis reports error
//   axisdata[2].Axis_Error: A-0-0021.09 -RD- Axis reports error
//   drive2: Real axis "Drive2" with axis number 2
ton_en_2(IN := b_enable_az_2 AND NOT axisdata[1].Axis_Error AND NOT axisdata[2].Axis_Error, PT := t#100ms); // TON
FB_2_power(Enable := ton_en_2.Q, Axis := drive2); // MC_Power

// NETWORK 10
//   axisdata[1].Axis_Power: A-0-0021.15 -RD- Axis has power on (AH_AF)
//   axisdata[2].Axis_Power: A-0-0021.15 -RD- Axis has power on (AH_AF)
// label: (*home drive2*)
b_home_az2_done := axisdata[1].Axis_Power AND axisdata[2].Axis_Power;

// NETWORK 11 (disabled)
//   axisdata[1].Axis_Power: A-0-0021.15 -RD- Axis has power on (AH_AF)
//   axisdata[2].Axis_Power: A-0-0021.15 -RD- Axis has power on (AH_AF)
// label: (*home drive2*)
// b_home_az2_done := axisdata[1].Axis_Power AND axisdata[2].Axis_Power;

// NETWORK 12
//   FB_move_master_az: "MC_MoveAbsolute" is used to move the drive to a preset absolute position.
//   AxisData[1].rActualPosition_i: A-0-0100 -RD- Actual position
//   v_azimuth: Virtual axis "v_azimuth" with axis number 7
// label: (*move azimuth virtual axis to the position of driver 1*)
FB_move_master_az(
    Execute := b_home_az2_done,
    Position := AxisData[1].rActualPosition_i,
    Velocity := 999,
    Acceleration := 99,
    Deceleration := 99,
    Axis := v_azimuth); // MC_MoveAbsolute
b_M_az_done := FB_move_master_az.Done;

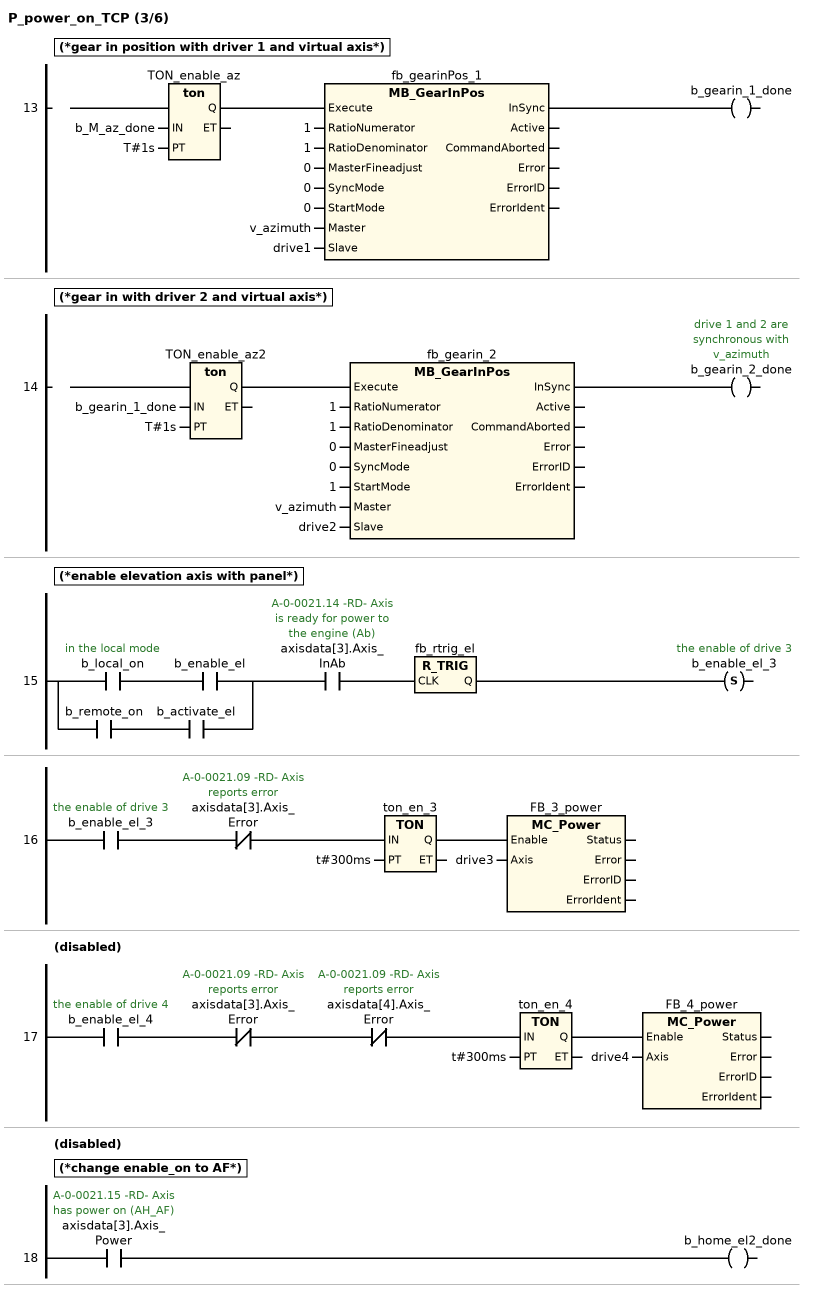
// NETWORK 13
//   fb_gearinPos_1: With "MB_GearInPos",it is possible to realize a motion of the slave axis which is phase synchronous to the master axis
//   v_azimuth: Virtual axis "v_azimuth" with axis number 7
//   drive1: Real axis "Drive1" with axis number 1
// label: (*gear in position with driver 1 and virtual axis*)
TON_enable_az(IN := b_M_az_done, PT := T#1s); // ton
fb_gearinPos_1(
    Execute := TON_enable_az.Q,
    RatioNumerator := 1,
    RatioDenominator := 1,
    MasterFineadjust := 0,
    SyncMode := 0,
    StartMode := 0,
    Master := v_azimuth,
    Slave := drive1); // MB_GearInPos
b_gearin_1_done := fb_gearinPos_1.InSync;

// NETWORK 14
//   v_azimuth: Virtual axis "v_azimuth" with axis number 7
//   drive2: Real axis "Drive2" with axis number 2
//   b_gearin_2_done: drive 1 and 2 are synchronous with v_azimuth
// label: (*gear in with driver 2 and virtual axis*)
TON_enable_az2(IN := b_gearin_1_done, PT := T#1s); // ton
fb_gearin_2(
    Execute := TON_enable_az2.Q,
    RatioNumerator := 1,
    RatioDenominator := 1,
    MasterFineadjust := 0,
    SyncMode := 0,
    StartMode := 1,
    Master := v_azimuth,
    Slave := drive2); // MB_GearInPos
b_gearin_2_done := fb_gearin_2.InSync;

// NETWORK 15
//   b_local_on: in the local mode
//   axisdata[3].Axis_InAb: A-0-0021.14 -RD- Axis is ready for power to the engine (Ab)
//   b_enable_el_3: the enable of drive 3
// label: (*enable elevation axis with panel*)
fb_rtrig_el(CLK := (b_local_on AND b_enable_el OR b_remote_on AND b_activate_el) AND axisdata[3].Axis_InAb); // R_TRIG
b_enable_el_3 S= fb_rtrig_el.Q;

// NETWORK 16
//   b_enable_el_3: the enable of drive 3
//   axisdata[3].Axis_Error: A-0-0021.09 -RD- Axis reports error
//   drive3: Real axis "Drive3" with axis number 3
ton_en_3(IN := b_enable_el_3 AND NOT axisdata[3].Axis_Error, PT := t#300ms); // TON
FB_3_power(Enable := ton_en_3.Q, Axis := drive3); // MC_Power

// NETWORK 17 (disabled)
//   b_enable_el_4: the enable of drive 4
//   axisdata[3].Axis_Error: A-0-0021.09 -RD- Axis reports error
//   axisdata[4].Axis_Error: A-0-0021.09 -RD- Axis reports error
//   drive4: Real axis "Drive4" with axis number 4
// ton_en_4(IN := b_enable_el_4 AND NOT axisdata[3].Axis_Error AND NOT axisdata[4].Axis_Error, PT := t#300ms); // TON
// FB_4_power(Enable := ton_en_4.Q, Axis := drive4); // MC_Power

// NETWORK 18 (disabled)
//   axisdata[3].Axis_Power: A-0-0021.15 -RD- Axis has power on (AH_AF)
// label: (*change enable_on to AF*)
// b_home_el2_done := axisdata[3].Axis_Power;

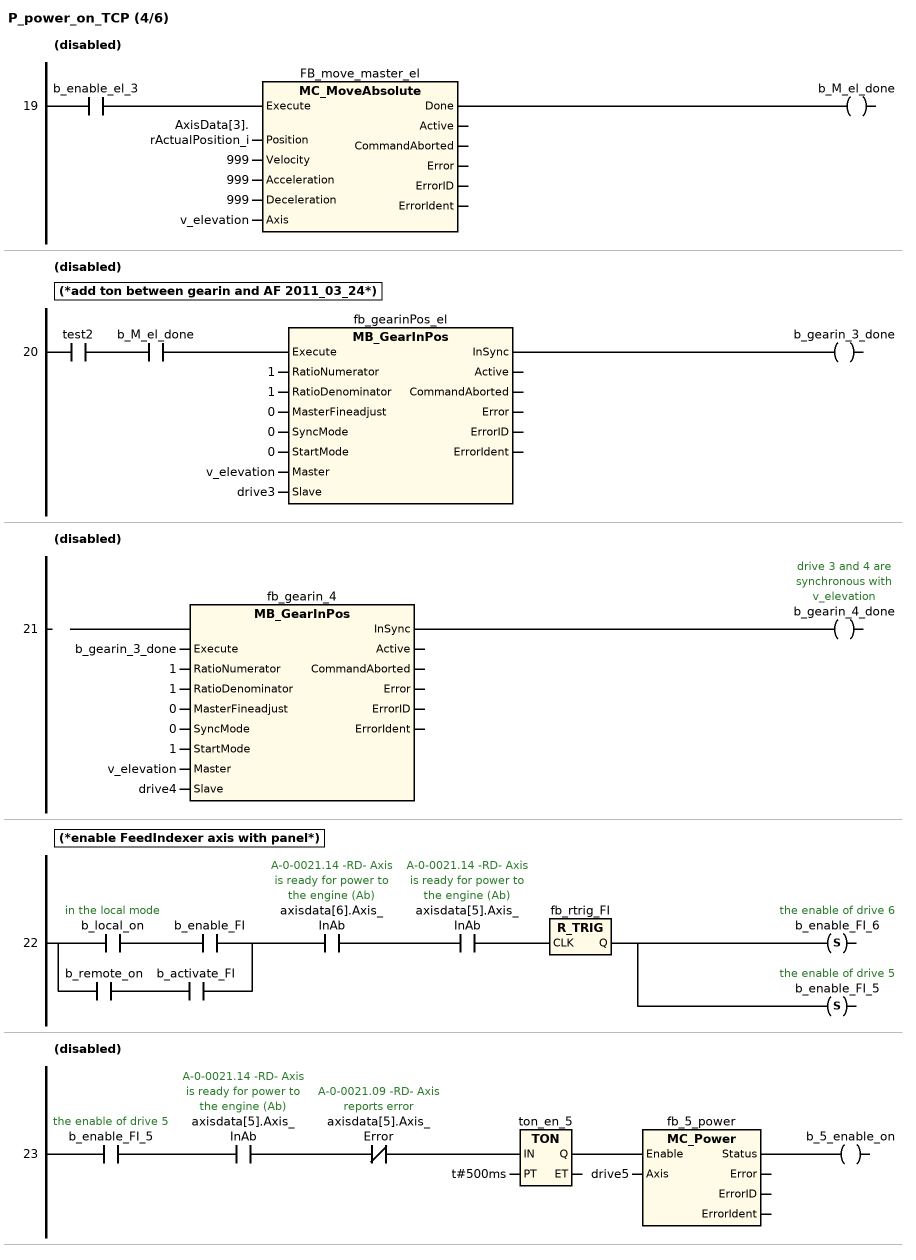
// NETWORK 19 (disabled)
//   AxisData[3].rActualPosition_i: A-0-0100 -RD- Actual position
//   v_elevation: Virtual axis "v_elevation" with axis number 8
// FB_move_master_el(
//     Execute := b_enable_el_3,
//     Position := AxisData[3].rActualPosition_i,
//     Velocity := 999,
//     Acceleration := 999,
//     Deceleration := 999,
//     Axis := v_elevation); // MC_MoveAbsolute
// b_M_el_done := FB_move_master_el.Done;

// NETWORK 20 (disabled)
//   fb_gearinPos_el: add 2011 06 09 to delete 1sec delay
//   v_elevation: Virtual axis "v_elevation" with axis number 8
//   drive3: Real axis "Drive3" with axis number 3
// label: (*add ton between gearin and AF 2011_03_24*)
// fb_gearinPos_el(
//     Execute := test2 AND b_M_el_done,
//     RatioNumerator := 1,
//     RatioDenominator := 1,
//     MasterFineadjust := 0,
//     SyncMode := 0,
//     StartMode := 0,
//     Master := v_elevation,
//     Slave := drive3); // MB_GearInPos
// b_gearin_3_done := fb_gearinPos_el.InSync;

